(*************************** 647**************************************)
// Wyspa 647 - podajnik opakowań
QABPneumatic647ValveCoils[1].0 := P08_CapSorter.QbCapSorterDragActuator;     //[710, 5/3, wysunięcie wideł]
QABPneumatic647ValveCoils[1].1 := NOT P08_CapSorter.QbCapSorterDragActuator;					
QABPneumatic647ValveCoils[1].2 := P08_CapSorter.QbCapSorterDragLeadBefore1Actuator;    //[720, 5/3 , wysunięcie prowaadzenie ]
QABPneumatic647ValveCoils[1].3 := NOT P08_CapSorter.QbCapSorterDragLeadBefore1Actuator;
QABPneumatic647ValveCoils[1].4 := P08_CapSorter.QbCapSorterStoperActuator;   //[730, 5/2, wysunięcie amortyzatora]
QABPneumatic647ValveCoils[1].5;
QABPneumatic647ValveCoils[1].6 := P08_CapSorter.QbCapSorterDragLeadAfter1Actuator;
QABPneumatic647ValveCoils[1].7 := NOT P08_CapSorter.QbCapSorterDragLeadAfter1Actuator;
QABPneumatic647ValveCoils[2].0;
QABPneumatic647ValveCoils[2].1 := QbBlowBeforeGripperScrewer;//nie ma
QABPneumatic647ValveCoils[2].2 := QbGripperScrewerGateBeforeActuator; //nie ma
QABPneumatic647ValveCoils[2].3;
(*********************Koniec 647 **************************************)

(*************************** 641 **************************************)
QABPneumaticPI641ValveCoils[1].0	:= NOT P01_pucksInserter.QbPucksInserterHammer;
QABPneumaticPI641ValveCoils[1].1	:= P01_pucksInserter.QbPucksInserterHammer;					
QABPneumaticPI641ValveCoils[1].2	:= P01_pucksInserter.QbPucksInserterTray;
QABPneumaticPI641ValveCoils[1].3	:= NOT P01_pucksInserter.QbPucksInserterTray;
QABPneumaticPI641ValveCoils[1].4	:= NOT P01_pucksInserter.QbPucksInserterGate1;
QABPneumaticPI641ValveCoils[1].5	:=  P01_pucksInserter.QbPucksInserterGate1;
QABPneumaticPI641ValveCoils[1].6	:=  NOT P01_pucksInserter.QbPucksInserterGate2;
QABPneumaticPI641ValveCoils[1].7	:=  P01_pucksInserter.QbPucksInserterGate2;
QABPneumaticPI641ValveCoils[2].0 	:=  NOT P01_pucksInserter.QbPucksInserterFormGate;
QABPneumaticPI641ValveCoils[2].1	:=  P01_pucksInserter.QbPucksInserterFormGate;
QABPneumaticPI641ValveCoils[2].2	:=  NOT P01_pucksInserter.QbPucksInserterFormPositioning;
QABPneumaticPI641ValveCoils[2].3  :=  FALSE;//:= NOT P01_PucksInserter.QbPucksInserterPushTable_Gate;    //Vasyl 27.05 [670, 5/2 Szlabany stołu podającego]                    
QABPneumaticPI641ValveCoils[2].4	;//:= 	P01_PucksInserter.QbPucksInserterPushTable_Gate;	
QABPneumaticPI641ValveCoils[2].5;
QABPneumaticPI641ValveCoils[2].6	;//:= P01_PucksInserter.QbPucksInserterPushTable_Pushers; //Vasyl 04.08   [5/2 Popychacze stołu podającego]
QABPneumaticPI641ValveCoils[2].7;
(*********************Koniec 641 **************************************)
END_ACTION

ACTION aVTEM:
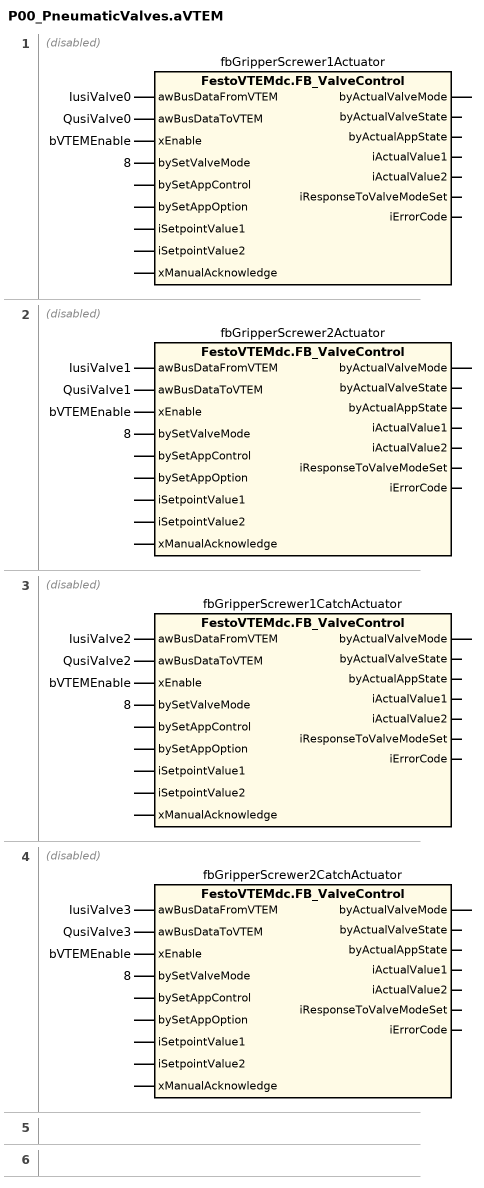
// NETWORK 1 (disabled)
// fbGripperScrewer1Actuator(
//     awBusDataFromVTEM := IusiValve0,
//     awBusDataToVTEM := QusiValve0,
//     xEnable := bVTEMEnable,
//     bySetValveMode := 8); // FestoVTEMdc.FB_ValveControl

// NETWORK 2 (disabled)
// fbGripperScrewer2Actuator(
//     awBusDataFromVTEM := IusiValve1,
//     awBusDataToVTEM := QusiValve1,
//     xEnable := bVTEMEnable,
//     bySetValveMode := 8); // FestoVTEMdc.FB_ValveControl

// NETWORK 3 (disabled)
// fbGripperScrewer1CatchActuator(
//     awBusDataFromVTEM := IusiValve2,
//     awBusDataToVTEM := QusiValve2,
//     xEnable := bVTEMEnable,
//     bySetValveMode := 8); // FestoVTEMdc.FB_ValveControl

// NETWORK 4 (disabled)
// fbGripperScrewer2CatchActuator(
//     awBusDataFromVTEM := IusiValve3,
//     awBusDataToVTEM := QusiValve3,
//     xEnable := bVTEMEnable,
//     bySetValveMode := 8); // FestoVTEMdc.FB_ValveControl

// NETWORK 5

// NETWORK 6
END_ACTION

ACTION aVTEMSignals:
// Wszystkie od 1 do 8 bar
(*
(********VTEM 0********)
(***     F[N]=p[bar]*14,8[N/bar] ************) // od 1,5kg do 12kg
IF lrGripperScrewerPressure = 0 					THEN	lrGripperScrewerPressure := 2; 						END_IF;
IF lrGripperScrewerPressureExhaustLevel < 10	THEN	lrGripperScrewerPressureExhaustLevel := 10;		END_IF;
fbGripperScrewer1Actuator.iSetpointValue2 := (**Smbar Setpoint sir supply pressure during travel**)
ABS(LREAL_TO_INT(((lrGripperScrewerPressure*10)/14.8)*1000));
IF fbGripperScrewer1Actuator.iSetpointValue2 >8000 THEN
	fbGripperScrewer1Actuator.iSetpointValue2 := 8000;
END_IF
IF fbGripperScrewer1Actuator.iSetpointValue2 >8000 THEN
	fbGripperScrewer1Actuator.iSetpointValue2 := 8000;
END_IF
IF P10_GripperScrewer.QbGripperScrewer1Actuator THEN(**Włączanie zaworu**)
	fbGripperScrewer1Actuator.bySetAppControl	:= 2;
	fbGripperScrewer1Actuator.iSetpointValue1	:= LREAL_TO_INT(lrGripperScrewerPressureExhaustLevel*100);//10000;(**Setpoint opening degree axhaust air flow control**)
ELSE
	fbGripperScrewer1Actuator.bySetAppControl	:= 3;
	fbGripperScrewer1Actuator.iSetpointValue1	:= 10000;(**Setpoint opening degree axhaust air flow control**)
END_IF	
IF fbGripperScrewer1Actuator.iResponseToValveModeSet = 1037 (*Acknoledge_needed*) THEN
	fbGripperScrewer1Actuator.xManualAcknowledge := TRUE;	ELSE
	fbGripperScrewer1Actuator.xManualAcknowledge := FALSE;	END_IF
	
	
(********VTEM 1********)
(***     F[N]=p[bar]*14,8[N/bar] ************) // od 1,5kg do 12kg
IF lrGripperScrewerPressure = 0 					THEN	lrGripperScrewerPressure := 2; 						END_IF;
IF lrGripperScrewerPressureExhaustLevel < 10	THEN	lrGripperScrewerPressureExhaustLevel := 10;		END_IF;
fbGripperScrewer2Actuator.iSetpointValue2 := (**Smbar Setpoint sir supply pressure during travel**)
ABS(LREAL_TO_INT(((lrGripperScrewerPressure*10)/14.8)*1000));
IF fbGripperScrewer2Actuator.iSetpointValue2 >8000 THEN
	fbGripperScrewer2Actuator.iSetpointValue2 := 8000;
END_IF
IF fbGripperScrewer2Actuator.iSetpointValue2 >8000 THEN
	fbGripperScrewer2Actuator.iSetpointValue2 := 8000;
END_IF
IF P10_GripperScrewer.QbGripperScrewer2Actuator THEN(**Włączanie zaworu**)
	fbGripperScrewer2Actuator.bySetAppControl	:= 2;
	fbGripperScrewer2Actuator.iSetpointValue1	:= LREAL_TO_INT(lrGripperScrewerPressureExhaustLevel*100);(**Setpoint opening degree axhaust air flow control**)
ELSE
	fbGripperScrewer2Actuator.bySetAppControl	:= 3;
	fbGripperScrewer2Actuator.iSetpointValue1	:= 10000;(**Setpoint opening degree axhaust air flow control**)
END_IF	
IF fbGripperScrewer2Actuator.iResponseToValveModeSet = 1037 (*Acknoledge_needed*) THEN
	fbGripperScrewer2Actuator.xManualAcknowledge := TRUE;	ELSE
	fbGripperScrewer2Actuator.xManualAcknowledge := FALSE;	END_IF
	
	
(********VTEM 2********)
IF lrGripperScrewerPressure = 0 					THEN	lrGripperScrewerPressure := 3; 						END_IF;
IF (lrGripperScrewerCatchPressureExhaustLevel < 10)	THEN	lrGripperScrewerCatchPressureExhaustLevel := 10;		END_IF; // bylo <1000
fbGripperScrewer1CatchActuator.iSetpointValue2 := (**Smbar Setpoint sir supply pressure during travel**)
ABS(LREAL_TO_INT(((lrGripperScrewerPressure*10)/26.2)*1000));
IF fbGripperScrewer1CatchActuator.iSetpointValue2 >8000 THEN
	fbGripperScrewer1CatchActuator.iSetpointValue2 := 8000;
END_IF
IF P10_GripperScrewer.QbGripperScrewer1CatchActuator THEN(**Włączanie zaworu**)
	fbGripperScrewer1CatchActuator.bySetAppControl	:= 1;
	fbGripperScrewer1CatchActuator.iSetpointValue1	:= LREAL_TO_INT((lrGripperScrewerCatchPressureExhaustLevel*15.5)-55);(**Setpoint opening degree axhaust air flow control**)
ELSE
	fbGripperScrewer1CatchActuator.bySetAppControl	:= 2;
	fbGripperScrewer1CatchActuator.iSetpointValue1	:= 10000;(**Setpoint opening degree axhaust air flow control**)
END_IF
IF fbGripperScrewer1CatchActuator.iResponseToValveModeSet = 1037 (*Acknoledge_needed*) THEN
	fbGripperScrewer1CatchActuator.xManualAcknowledge := TRUE;	ELSE
	fbGripperScrewer1CatchActuator.xManualAcknowledge := FALSE;	END_IF	
		
	
(********VTEM 3********)
IF lrGripperScrewerPressure = 0 					THEN	lrGripperScrewerPressure := 3; 						END_IF;
IF ((lrGripperScrewerCatchPressureExhaustLevel) < 10)	THEN	lrGripperScrewerCatchPressureExhaustLevel := 10;		END_IF; // było <1000 i 100000

fbGripperScrewer2CatchActuator.iSetpointValue2 := (**Smbar Setpoint sir supply pressure during travel**)
ABS(LREAL_TO_INT(((lrGripperScrewerPressure*10)/26.2)*1000));
IF fbGripperScrewer2CatchActuator.iSetpointValue2 >8000 THEN
	fbGripperScrewer2CatchActuator.iSetpointValue2 := 8000;
END_IF
IF P10_GripperScrewer.QbGripperScrewer2CatchActuator THEN(**Włączanie zaworu**)
	fbGripperScrewer2CatchActuator.bySetAppControl	:= 1;
	fbGripperScrewer2CatchActuator.iSetpointValue1	:= LREAL_TO_INT((lrGripperScrewerCatchPressureExhaustLevel*15.5)-55);(**Setpoint opening degree axhaust air flow control**)
ELSE
	fbGripperScrewer2CatchActuator.bySetAppControl	:= 2;
	fbGripperScrewer2CatchActuator.iSetpointValue1	:= 10000;(**Setpoint opening degree axhaust air flow control**)
END_IF
IF fbGripperScrewer2CatchActuator.iResponseToValveModeSet = 1037 (*Acknoledge_needed*) THEN
	fbGripperScrewer2CatchActuator.xManualAcknowledge := TRUE;	ELSE
	fbGripperScrewer2CatchActuator.xManualAcknowledge := FALSE;	END_IF	
			
	
*)
END_ACTION

END_PROGRAM

// ---- POUs/FB/Various/FB_4_20mA_TO_INT.TcPOU
FUNCTION_BLOCK FB_4_20mA_TO_INT
VAR_INPUT
	iIN		:	INT;	(*Zmienna skalowana*)
	rXmin	:	REAL;	(*Dolny zakres zmiennej przeskalowanej*)
	rXmax	:	REAL;	(*Górny zakres zmiennej przeskalowanej*)
	rYmin	:	REAL;	(*Dolny zakres zmiennej skalowanej*)
	rYmax	:	REAL;	(*Górny zakres zmiennej skalowanej*)
END_VAR
VAR_OUTPUT
	bError  :	BOOL;
	iOUT	:	INT;	(*Zmienna skalowana*)
END_VAR
VAR
	rfA		:	REAL;	
	rfB		:	REAL;	
	rfC		:	REAL;	
END_VAR


rfA := (rYmax-rYmin)/(rXmax-rXmin);
rfB := (INT_TO_REAL(iIN)-rXmin);
rfC := rYmin;
iOUT := REAL_TO_INT(rfA*rfB+rfC);

IF iIN < rXmin-1 OR iIN>rXmax+1 THEN
	bError	:= TRUE;
	iOUT	:= REAL_TO_INT(rYmax);
ELSE
	bError	:= FALSE;
END_IF

END_FUNCTION_BLOCK

// ---- POUs/FB/Conversions/BitOriented/F_2Bytes_To_Word.TcPOU
(****************************************************************************************)
(*							Beckhoff Automation Poland									*)
(*								F_2Bytes_To_Word v1.0									*)
(*									15.02.2010											*)
(*		Funkcja tworząca zmienną typu WORD z dwóch zmiennych typu BYTE					*)
(*______________________________________________________________________________________*)
FUNCTION F_2Bytes_To_Word : WORD
VAR_INPUT
	byHigh	:	BYTE;
	byLow	:	BYTE;
END_VAR
VAR
END_VAR

F_2Bytes_To_Word := byHigh;
F_2Bytes_To_Word := SHL(F_2Bytes_To_Word,8);
F_2Bytes_To_Word := F_2Bytes_To_Word + byLow;

END_FUNCTION

// ---- POUs/P10_GripperScrewer.TcPOU
(*
Nazwa:			P10_GripperScrewer
Opis:			Stacja zakecarki szczekowej
Wersja:			v0.2
Data:			2018-10-10
Autor:			DP
Urzadzenia:		
Konfiguracja:	
Info:
- aktualizacja bloków
*)
PROGRAM P10_GripperScrewer
VAR_INPUT
	IlrGripperScrewer1HeightCV 							: LREAL;		// Wejscie czujnika dociśnięcia
	IlrGripperScrewer2HeightCV 							: LREAL;		// Wejscie czujnika dociśnięcia
	IbGripperScrewer1CatchActuatorSensor 		  		: BOOL;			// Czujnik otwarcia 
	IbGripperScrewer2CatchActuatorSensor 		  		: BOOL;			// Czujnik otwarcia
	{warning {'dodac czujniki otwarcia chwytaka'}
	IbGripperScrewersThirdFormCheckFormSensor	 	AT %I*	: BOOL; 		// Czujnik dojazdu 3 formatki
	IbGripperScrewersBeforeThirdFormCheckFormSensor	AT %I* 	: BOOL; 		// Czujnik po 3 formatce
	IbGripperScrewersSixthFormCheckFormSensor 		AT %I*	: BOOL;			//Czujnik dojazdu 6 formatki
	IbGripperScrewersDragUpSensor 			 		AT %I*	: BOOL;			// Czujnik
	IbGripperScrewersDragDownSensor 			 	AT %I*	: BOOL;			// Czujnik
	IbGripperScrewersDragHomingSensor 				AT %I*	: BOOL;			// Czujnik bazowania
	IbGripperScrewersDragLeadBefore1UpSensor 		AT %I* 	: BOOL;			// Czujnik
	IbGripperScrewersDragLeadBefore2UpSensor 		AT %I* 	: BOOL;			// Czujnik
END_VAR
VAR
	tonSimu1											:	ton;
	tonSimu2											:	ton;
	//ZMIENNE ZAKRĘCARKI	
	fb2GripperScrewer1									: FB_2GripperScrewers; 				// Blok funkcyjny sterujący zakręcarką szczękową
	fb2GripperScrewerNew1								: FB_2GripperScrewers_New; 			// Blok funkcyjny sterujący zakręcarką szczękową
	eGripperScrewer1State								: E_Station;						// Stan zakręcarki
	eGripperScrewer1RunningState						: E_GripperScrewer;				// Stan zakręcarki
	fb2GripperScrewer2									: FB_2GripperScrewers; 				// Blok funkcyjny sterujący zakręcarką szczękową
	fb2GripperScrewerNew2								: FB_2GripperScrewers_New; 			// Blok funkcyjny sterujący zakręcarką szczękową
	eGripperScrewer2State								: E_Station;						// Stan zakręcarki
	eGripperScrewer2RunningState						: E_GripperScrewer;				// Stan zakręcarki
	fbGripperScrewer1State								: FB_State;
	fbGripperScrewer2State								: FB_State;
	                                        		
	//Zmienne chwytaka                      		
	fbGripperScrewer1CatchStation						: FB_CatchStation;			// Blok funkcyjny sterowania chwytaka zakręcarką szczękową
	eGripperScrewer1CatchState							: E_Station;                  // Stan chwytaka stabilizujšcego pod zakręcarkš
	eGripperScrewer1CatchRunningState					: E_CatchStationState;        // Stan chwytaka stabilizujšcego pod zakręcarkš
	fbGripperScrewer1CatchState							: FB_State;
	
	//WEJSCIA WYJSCIA
	QbGripperScrewer1Actuator							: BOOL; 				// Sterowanie siłownikiem chwytaka zakrecarki szczękowej (Podłączenie do Bajtu sterującego wyspy)
	QnGripperScrewer1TorqueLimit 				AT %Q*	: UINT; 				// Ograniczenie momentu napędu zakręcarki szczękowej 
	QnGripperScrewer1ProportionalGain 			AT %Q*	: REAL; 				// Kp 
	IdiGripperScrewer1HeightCV 					AT %I*	: DINT;			// Wejscie czujnika dociśnięcia
	IrGripperScrewer1ActualMotorTemperature 	AT %I*	: REAL; 				// Aktualna temperatura silnika zakręcarki
	
	//Chwytak zakecarki szczękowej
	QbGripperScrewer1CatchHeightUpCmd 			AT %Q*	: BOOL; 				// Wyjście sterujące podnośnikiem siłownika stabilizującego pod zakręcarką szczękową, Silnik w górę
	QbGripperScrewer1CatchHeightDownCmd 		AT %Q*	: BOOL; 				// Wyjście sterujące podnośnikiem siłownika stabilizującego pod zakręcarką szczękową, Silnik w dół
	QbGripperScrewer1CatchActuator						: BOOL; 				// Sterowanie siłownikiem chwytaka stabilizującego pod zakręcarką szczękową (Podłączenie do Bajtu sterującego wyspy)
	IbGripperScrewer1CatchHeightEncoderPulse 	AT %I*  : BOOL;					// Wejście impulsów enkodera podnośnika chwytaka pod zakręcarką
	
	tofTimerGripperScrewer1Enable						: TOF;
	rtbGripperScrewer12EnableShow						: R_TRIG;
	ftbGripperScrewer12EnableShow						: F_TRIG;	
	rtEnable1											: R_TRIG;
	
	(*Wykres dozowania*)
	fbGripperScrewer1Chart								: FB_WriteDataToArrayString;
	fbGripperScrewer1StChart							: FB_WriteDataToArrayOfArrays;
	fbGripperScrewer2StChart							: FB_WriteDataToArrayOfArrays;
	rtStartGripper1Screwing								: R_TRIG;
	lrGripperScrewer1AxisStartPosition					: LREAL;
	nCountTest555										: INT;
	nCountTest556										: INT;
	nCountTest557										: INT;
	nGripperScrewer1AdjustingDialog						: INT;
	bGripperScrewer1AdjustTorqueDialog					: BOOL;
	nTstcount											: INT;

	//Zmienne chwytaka
	fbGripperScrewer2CatchStation						: FB_CatchStation;			// Blok funkcyjny sterowania chwytaka zakręcarką szczękową
	eGripperScrewer2CatchState							: E_Station;                  // Stan chwytaka stabilizujšcego pod zakręcarkš
	eGripperScrewer2CatchRunningState					: E_CatchStationState;        // Stan chwytaka stabilizujšcego pod zakręcarkš
	fbGripperScrewerCatch2State							: FB_State;
	
	
	//WEJSCIA WYJSCIA
	QbGripperScrewer2Actuator							: BOOL; 	(*Pneu*)		// Sterowanie siłownikiem chwytaka zakrecarki szczękowej (Podłączenie do Bajtu sterującego wyspy)
	QnGripperScrewer2TorqueLimit 				AT %Q*	: UINT; 	(*do driva*)	// Ograniczenie momentu napędu zakręcarki szczękowej 
	QnGripperScrewer2ProportionalGain 			AT %Q*	: REAL; 				// Kp 
	IrGripperScrewer2ActualMotorTemperature 	AT %I*	: REAL; 	(*do driva*)	// Aktualna temperatura silnika zakręcarki
	IdiGripperScrewer2HeightCV 					AT %I*	: DINT;			// Wejscie czujnika dociśnięcia
	IbGripperScrewersHeightEncoderSetCDone				AT %I*: BOOL;
	IudiGripperScrewersHeightEncoderCV          AT %I*: UDINT;
	QbGripperScrewersHeightEncoderSetC 			AT %Q*: BOOL;
	QudiGripperScrewersHeightEncoderSetCV       AT %Q*: UDINT;
	
	//Chwytak zakecarki szczękowej
	QbGripperScrewer2CatchHeightUpCmd 			AT %Q*	: BOOL; 			(*PLC.A19*)	 	// Wyjście sterujące podnośnikiem siłownika stabilizującego pod zakręcarką szczękową, Silnik w górę
	QbGripperScrewer2CatchHeightDownCmd 		AT %Q*	: BOOL; 		(*PLC.A19*)		// Wyjście sterujące podnośnikiem siłownika stabilizującego pod zakręcarką szczękową, Silnik w dół
	QbGripperScrewer2CatchActuator						: BOOL; 					(*Pneu*)		// Sterowanie siłownikiem chwytaka stabilizującego pod zakręcarką szczękową (Podłączenie do Bajtu sterującego wyspy)
	IbGripperScrewer2CatchHeightEncoderPulse  	AT %I*  : BOOL;	(*PLC.A15*)		// Wejście impulsów enkodera podnośnika chwytaka pod zakręcarką

	tofTimerGripperScrewer2Enable						: TOF;


	(*Wykres dozowania*)
	fbGripperScrewer2Chart								: FB_WriteDataToArrayString;
	rtStartGripper2Screwing								: R_TRIG;
	lrGripperScrewer2AxisStartPosition					: LREAL;
	
	(*******PRZECIAGANIE**********)
	fbGripperScrewersDragStation						: FB_FormsDragStepper;
	eFormsDragingPneumaticState							: E_Station;						// Stan zakręcarki
	eFormsDragingPneuamticRunningState					: E_DragStationState;			// Stan zakręcarki
	fbFormsDragingPneumaticState						: FB_State;
	
	//WEJSCIA I WYJSCIA SPRZETOW
	QbGripperScrewersDragLeadBefore1Actuator        	:BOOL;						// Siłownikiem prowadzenia przed 1(1 faza)
	QbGripperScrewersDragActuator                	  	:BOOL;						// Siłownikiem przeciągania (1 faza)
	
	tDelayCatchValve									: TIME;
	tonGriperScrewerCatch1ValveOpenSensor				: TON;
	tonGriperScrewerCatch2ValveOpenSensor				: TON;
		
	(*kasowanie offsetu*)
	tonGripperScrewer1SetPositionOffsetReset			: TON;
	tonGripperScrewer2SetPositionOffsetReset			: TON;

	(*Filtrowqanie momentu*)
	fbFilterTorque1						: FB_FilterEx;					// Bloczek do filtrowania (*NOWE*)
	rFilteredTorque1Value				: REAL;							// Zmiena odfiltrowana (*NOWE*)
	fbFilterTorque2						: FB_FilterEx;					// Bloczek do filtrowania (*NOWE*)
	rFilteredTorque2Value				: REAL;							// Zmiena odfiltrowana (*NOWE*)
	
	(*Szukanie gwintu*)
	lrGripperScrewerPushingCapPositionTemp	:	LREAL;
	lrGripperScrewerScrewingCapPositionTemp	:	LREAL;
	rtGripperScrewerFindScrewAdjust			:	R_TRIG;
	rtGripperScrewerOption5					:	R_TRIG;
	iGripperScrewerFindScrewAdjust			:	INT;
	
	(*smieci*)
	btemp												: BOOL;
	atemp1												: AXIS_REF;
	atemp2												: AXIS_REF;
	
	(*inne*)
	bSimulationGripper									: BOOL;

	tofTimerGripperScrewer1Catch: TOF;
	tofTimerGripperScrewer2Catch: TOF;
	
//dodatkowa obsługa stopera formatek przy dojeździe 
	

	//tpStoperTimerOn							:TP;	// timer do generowania impulsu
	//fbStoperSensorDelay						:FB_InputFilter;	// filtr do generowania sygnału 
	//tofQbGripperScrewerStoperActuator		:TOF;
	//lrStoperPosition: LREAL;
	bTestZakrecania: BOOL;
	
	rtfb2GripperScrewer1Done: R_TRIG;
	rtfb2GripperScrewer2Done: R_TRIG;	

	iGripperScrewer1Info1 : INT;
	iGripperScrewer2Info1 : INT;
	iGripperScrewer1NoWarningInRow : INT;
	iGripperScrewer2NoWarningInRow : INT;	
	bGripperScrewer1ChangeRubbers :BOOL;
	bGripperScrewer2ChangeRubbers :BOOL;	
	tonbGripperScrewer1ChangeRubbers: TON;
	tonbGripperScrewer2ChangeRubbers: TON;	
	
	//ManualStoper
	rtManualMode	: R_TRIG;
	ftManualMode	: F_TRIG;	
	bGripperScrewerStoperActuatorLastState	:BOOL;
	
	

	
END_VAR

(**Symulacja czujników otwarcia-zamknięcia chwytaka***)

tDelayCatchValve														:=T#50MS;

tonGriperScrewerCatch1ValveOpenSensor(IN:= NOT QbGripperScrewer1CatchActuator, PT:=tDelayCatchValve);
tonGriperScrewerCatch2ValveOpenSensor(IN:= NOT QbGripperScrewer2CatchActuator, PT:=tDelayCatchValve);
aStoper();
aDraging();
aCatch();
aLimits();
aFilter();
aGripperScrewerEnable();
aGripperScrewer();			//Nowa wersja zakrecarek STARA aGripperScrewer();
aGripperScrewerChartHMI();
aGripperScrewerDialogBox();
aGripperScrewerWarnings();
aFindScrewAdjust();
aInfo();

(***Skalownaie wartości zadanej na 1-100%************)
IF lrBottleDragingStationVelocity <50 THEN
	lrBottleDragingStationVelocity	:= 50;
END_IF 

(*** SKALOWANIE WARTOŚCI ZAKRĘCANIA Z Nm na % ***)
IF iPackageCapDiameter = 0 THEN
	iPackageCapDiameter 												:= 20;
END_IF

VIS.iPackageCapDiameterShow;
fb2GripperScrewer1.iScrewer1SetTorque 									:= LREAL_TO_INT((lrGripperScrewingTightTorque/1.5)*100);
fb2GripperScrewer2.iScrewer1SetTorque 									:= LREAL_TO_INT((lrGripperScrewing2TightTorque/1.5)*100);

(*** KONIEC SKALOWANIE WARTOŚCI ZAKRĘCANIA Z Nm na % ***)

(**** SKALOWANIE CZUJNIKOW WYSOKOSCI***)
IdiGripperScrewer1HeightCV;
//fb2GripperScrewer1.lrSpringHeightCV:= (IdiGripperScrewer1HeightCV *-1 ) + 110000;
//fb2GripperScrewer1.lrSpringHeightCV:= TO_LREAL(IdiGripperScrewer1HeightCV) /(-1000.0)+52.5; 
//

IdiGripperScrewer2HeightCV;
//fb2GripperScrewer2.lrSpringHeightCV:= (IdiGripperScrewer2HeightCV *-1 ) + 110000;
//fb2GripperScrewer2.lrSpringHeightCV:= TO_LREAL(IdiGripperScrewer2HeightCV) /(-1000.0)+52.1; 


(* BAZOWANIE - ZMIAN*)

tofTimerGripperScrewer1Catch(IN:=bGripperScrewer1Enable (*AND NOT bChangeover*), PT:=T#8S); 
tofTimerGripperScrewer2Catch(IN:=bGripperScrewer2Enable (*AND NOT bChangeover*), PT:=T#8S); 

rtEnable1(CLK:=fb2GripperScrewer1.bEnable1 OR fb2GripperScrewer2.bEnable1 ,Q=>);

VIS.lrGripperScrewer1LiftActPos											:= aGripperScrewer1LiftAxisRef.NcToPlc.ActPos;
VIS.lrGripperScrewer2LiftActPos											:= aGripperScrewer2LiftAxisRef.NcToPlc.ActPos;


IF rtEnable1.Q AND (P00_PackML.fbPMLAuto.ePMLState = E_PMLState.ePMLState_IDLE OR P00_PackML.fbPMLAuto.ePMLState = E_PMLState.ePMLState_EXECUTE)  THEN
	VIS.bGripperScrewerCatchHeightSet									:= TRUE;
	nCountTest555														:= nCountTest555+1;
ELSIF (fbGripperScrewer1CatchStation.eState=E_Station.eHomingDone AND fbGripperScrewer2CatchStation.eState=E_Station.eHomingDone)  AND fb2GripperScrewer1.eState=E_Station.eHomingDone AND fb2GripperScrewer2.eState=E_Station.eHomingDone THEN
	VIS.bGripperScrewerCatchHeightSet									:= FALSE;
	
ELSIF (fbGripperScrewer1CatchStation.eState=E_Station.eHomingDone AND fbGripperScrewer2CatchStation.eState=E_Station.eHomingDone)  THEN
	VIS.bGripperScrewerHeightSet										:= TRUE;
	
ELSIF (fb2GripperScrewer1.eState=E_Station.eHomingDone AND fb2GripperScrewer2.eState=E_Station.eHomingDone) OR VIS.bErrorOccure THEN
 	VIS.bGripperScrewerHeightSet										:= FALSE;
	nCountTest556														:= nCountTest556+1;
	
ELSIF (fbGripperScrewer1CatchStation.eState=E_Station.eHomingDone AND fbGripperScrewer2CatchStation.eState=E_Station.eHomingDone ) OR VIS.bErrorOccure  THEN
	VIS.bGripperScrewerCatchHeightSet									:= FALSE;
	VIS.bGripperScrewerHeightSet										:= FALSE;	
	nCountTest557														:= nCountTest557+1;
END_IF
(*KONIEC BAZOWANIE - ZMIANA*)


(********* GENEROWANIE STANU STACJI DO WIZKI**********)



fbGripperScrewer1State(
	eState																:= eGripperScrewer1State , 
	bRun																:= VIS.bGripperScrewer1Run OR VIS.bGripperScrewer1Run,	
	eGripperScrewerRunningState											:= eGripperScrewer1RunningState , 
	sStateDesc															=> VIS.sGripperScrewer1State,
	iState																=> VIS.iGripperScrewer1State);
fbGripperScrewer2State(
	eState																:= eGripperScrewer2State , 
	bRun																:= VIS.bGripperScrewer2Run OR VIS.bGripperScrewer2Run,	
	eGripperScrewerRunningState											:= eGripperScrewer2RunningState , 
	sStateDesc															=> VIS.sGripperScrewer2State,
	iState																=> VIS.iGripperScrewer2State);

fbGripperScrewer1CatchState(
	eState																:= eGripperScrewer1CatchState , 
	bRun																:= bGripperScrewer1Catch,	
	eCatchRunningState													:= eGripperScrewer1CatchRunningState , 
	sStateDesc															=> VIS.sGripperScrewerCatch1State,
	iState																=> VIS.iGripperScrewerCatch1State);	
	
fbGripperScrewerCatch2State(
	eState																:= eGripperScrewer2CatchState , 
	bRun																:= bGripperScrewer2Catch,	
	eCatchRunningState													:= eGripperScrewer2CatchRunningState , 
	sStateDesc															=> VIS.sGripperScrewerCatch2State,
	iState																=> VIS.iGripperScrewerCatch2State);	
	
fbFormsDragingPneumaticState(
	eState																:= eFormsDragingPneumaticState , 
	bRun																:= VIS.bBottleDragingStationRun,	
	eFormsDragingRunningState											:= eFormsDragingPneuamticRunningState , 
	sStateDesc															=> VIS.sBottleDragingStationState,
	iState																=> VIS.iBottleDragingStationState);	
	
		
(***** KONIEC GENEROWANIE STANU STACJI DO WIZKI*******)

(******* Wypracowanie sygnałów dla HMI *******)


VIS.bGripperScrewerCatch1ManualActuator;
(********KASOWANIE ROZKAZÓW CYKLI*********)
IF fb2GripperScrewer1.bCycleDone1 AND bManualMode THEN
	VIS.bGripperScrewer1Run 											:= FALSE;
END_IF
IF fb2GripperScrewer2.bCycleDone1 AND bManualMode THEN
	VIS.bGripperScrewer2Run 											:= FALSE;
END_IF

IF fbGripperScrewersDragStation.bCycleDone AND bManualMode THEN
	VIS.bBottleDragingStationRun 				:= FALSE;
	GVL.bBottleDragingStationPrepareRun			:= FALSE;
END_IF

(*Kasowanie offsetu po czasie*)
tonGripperScrewer1SetPositionOffsetReset(IN:=VIS.bGripperScrewer1SetPositionOffset, PT:=T#2S);
IF tonGripperScrewer1SetPositionOffsetReset.Q THEN
	VIS.bGripperScrewer1SetPositionOffset := FALSE;
END_IF
tonGripperScrewer2SetPositionOffsetReset(IN:=VIS.bGripperScrewer2SetPositionOffset, PT:=T#2S);
IF tonGripperScrewer2SetPositionOffsetReset.Q THEN
	VIS.bGripperScrewer2SetPositionOffset := FALSE;
END_IF
(*****KONIEC KASOWANIA ROZKAZÓW CYKLI*****)

aGripperScrewer1LiftAxisRef.NcToPlc.ActPos;
fb2GripperScrewer2.iToolHeight;

ACTION aCatch:
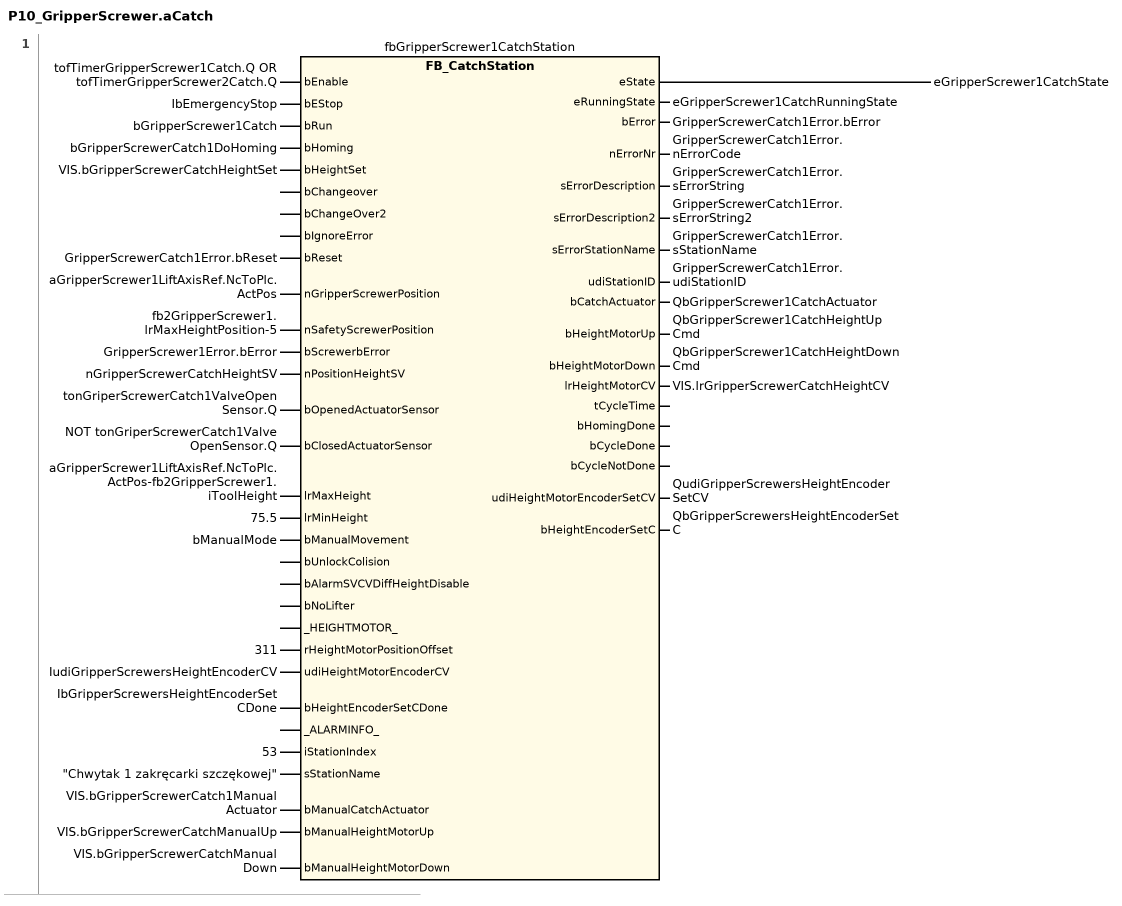
// NETWORK 1
fbGripperScrewer1CatchStation(
    bEnable := tofTimerGripperScrewer1Catch.Q OR tofTimerGripperScrewer2Catch.Q,
    bEStop := IbEmergencyStop,
    bRun := bGripperScrewer1Catch,
    bHoming := bGripperScrewerCatch1DoHoming,
    bHeightSet := VIS.bGripperScrewerCatchHeightSet,
    bReset := GripperScrewerCatch1Error.bReset,
    nGripperScrewerPosition := aGripperScrewer1LiftAxisRef.NcToPlc.ActPos,
    nSafetyScrewerPosition := fb2GripperScrewer1.lrMaxHeightPosition-5,
    bScrewerbError := GripperScrewer1Error.bError,
    nPositionHeightSV := nGripperScrewerCatchHeightSV,
    bOpenedActuatorSensor := tonGriperScrewerCatch1ValveOpenSensor.Q,
    bClosedActuatorSensor := NOT tonGriperScrewerCatch1ValveOpenSensor.Q,
    lrMaxHeight := aGripperScrewer1LiftAxisRef.NcToPlc.ActPos-fb2GripperScrewer1.iToolHeight,
    lrMinHeight := 75.5,
    bManualMovement := bManualMode,
    rHeightMotorPositionOffset := 311,
    udiHeightMotorEncoderCV := IudiGripperScrewersHeightEncoderCV,
    bHeightEncoderSetCDone := IbGripperScrewersHeightEncoderSetCDone,
    iStationIndex := 53,
    sStationName := "Chwytak 1 zakręcarki szczękowej",
    bManualCatchActuator := VIS.bGripperScrewerCatch1ManualActuator,
    bManualHeightMotorUp := VIS.bGripperScrewerCatchManualUp,
    bManualHeightMotorDown := VIS.bGripperScrewerCatchManualDown,
    eRunningState => eGripperScrewer1CatchRunningState,
    bError => GripperScrewerCatch1Error.bError,
    nErrorNr => GripperScrewerCatch1Error.nErrorCode,
    sErrorDescription => GripperScrewerCatch1Error.sErrorString,
    sErrorDescription2 => GripperScrewerCatch1Error.sErrorString2,
    sErrorStationName => GripperScrewerCatch1Error.sStationName,
    udiStationID => GripperScrewerCatch1Error.udiStationID,
    bCatchActuator => QbGripperScrewer1CatchActuator,
    bHeightMotorUp => QbGripperScrewer1CatchHeightUpCmd,
    bHeightMotorDown => QbGripperScrewer1CatchHeightDownCmd,
    lrHeightMotorCV => VIS.lrGripperScrewerCatchHeightCV,
    udiHeightMotorEncoderSetCV => QudiGripperScrewersHeightEncoderSetCV,
    bHeightEncoderSetC => QbGripperScrewersHeightEncoderSetC); // FB_CatchStation
eGripperScrewer1CatchState := fbGripperScrewer1CatchStation.eState;

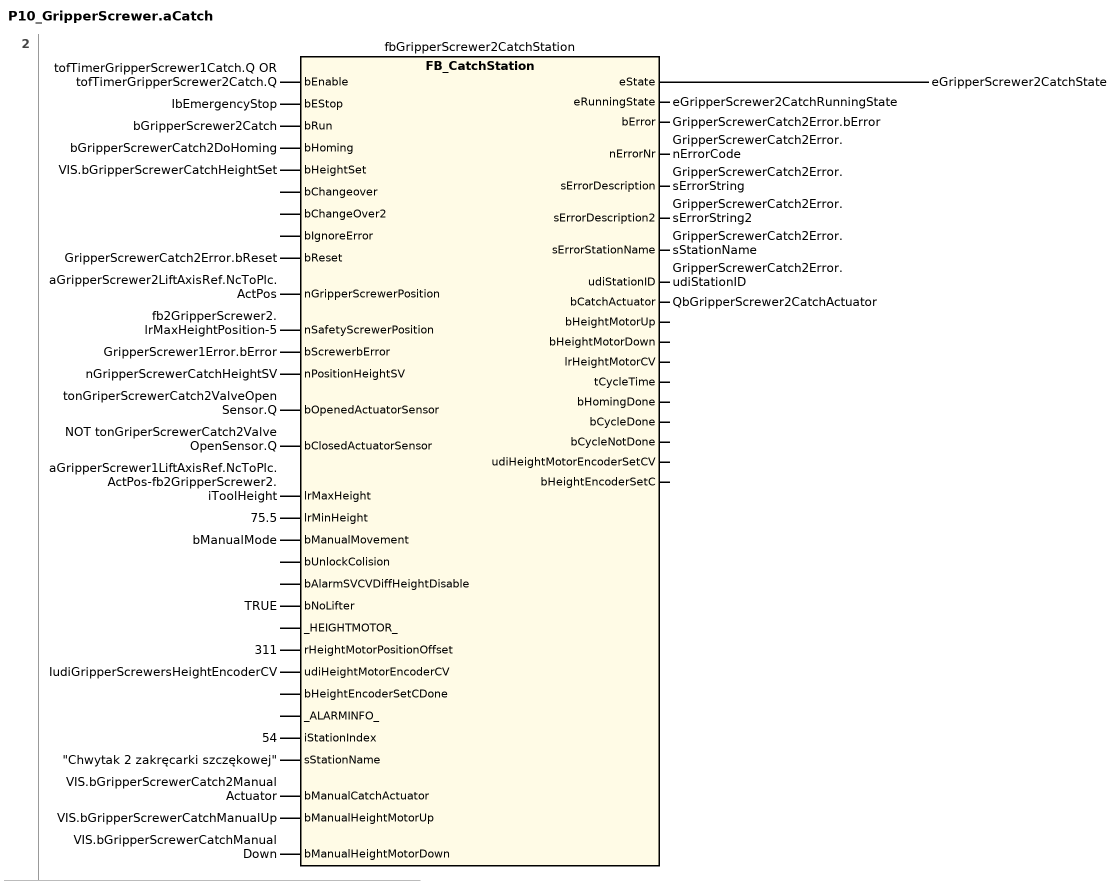
// NETWORK 2
fbGripperScrewer2CatchStation(
    bEnable := tofTimerGripperScrewer1Catch.Q OR tofTimerGripperScrewer2Catch.Q,
    bEStop := IbEmergencyStop,
    bRun := bGripperScrewer2Catch,
    bHoming := bGripperScrewerCatch2DoHoming,
    bHeightSet := VIS.bGripperScrewerCatchHeightSet,
    bReset := GripperScrewerCatch2Error.bReset,
    nGripperScrewerPosition := aGripperScrewer2LiftAxisRef.NcToPlc.ActPos,
    nSafetyScrewerPosition := fb2GripperScrewer2.lrMaxHeightPosition-5,
    bScrewerbError := GripperScrewer1Error.bError,
    nPositionHeightSV := nGripperScrewerCatchHeightSV,
    bOpenedActuatorSensor := tonGriperScrewerCatch2ValveOpenSensor.Q,
    bClosedActuatorSensor := NOT tonGriperScrewerCatch2ValveOpenSensor.Q,
    lrMaxHeight := aGripperScrewer1LiftAxisRef.NcToPlc.ActPos-fb2GripperScrewer2.iToolHeight,
    lrMinHeight := 75.5,
    bManualMovement := bManualMode,
    bNoLifter := TRUE,
    rHeightMotorPositionOffset := 311,
    udiHeightMotorEncoderCV := IudiGripperScrewersHeightEncoderCV,
    iStationIndex := 54,
    sStationName := "Chwytak 2 zakręcarki szczękowej",
    bManualCatchActuator := VIS.bGripperScrewerCatch2ManualActuator,
    bManualHeightMotorUp := VIS.bGripperScrewerCatchManualUp,
    bManualHeightMotorDown := VIS.bGripperScrewerCatchManualDown,
    eRunningState => eGripperScrewer2CatchRunningState,
    bError => GripperScrewerCatch2Error.bError,
    nErrorNr => GripperScrewerCatch2Error.nErrorCode,
    sErrorDescription => GripperScrewerCatch2Error.sErrorString,
    sErrorDescription2 => GripperScrewerCatch2Error.sErrorString2,
    sErrorStationName => GripperScrewerCatch2Error.sStationName,
    udiStationID => GripperScrewerCatch2Error.udiStationID,
    bCatchActuator => QbGripperScrewer2CatchActuator); // FB_CatchStation
eGripperScrewer2CatchState := fbGripperScrewer2CatchStation.eState;
END_ACTION

ACTION aDraging:
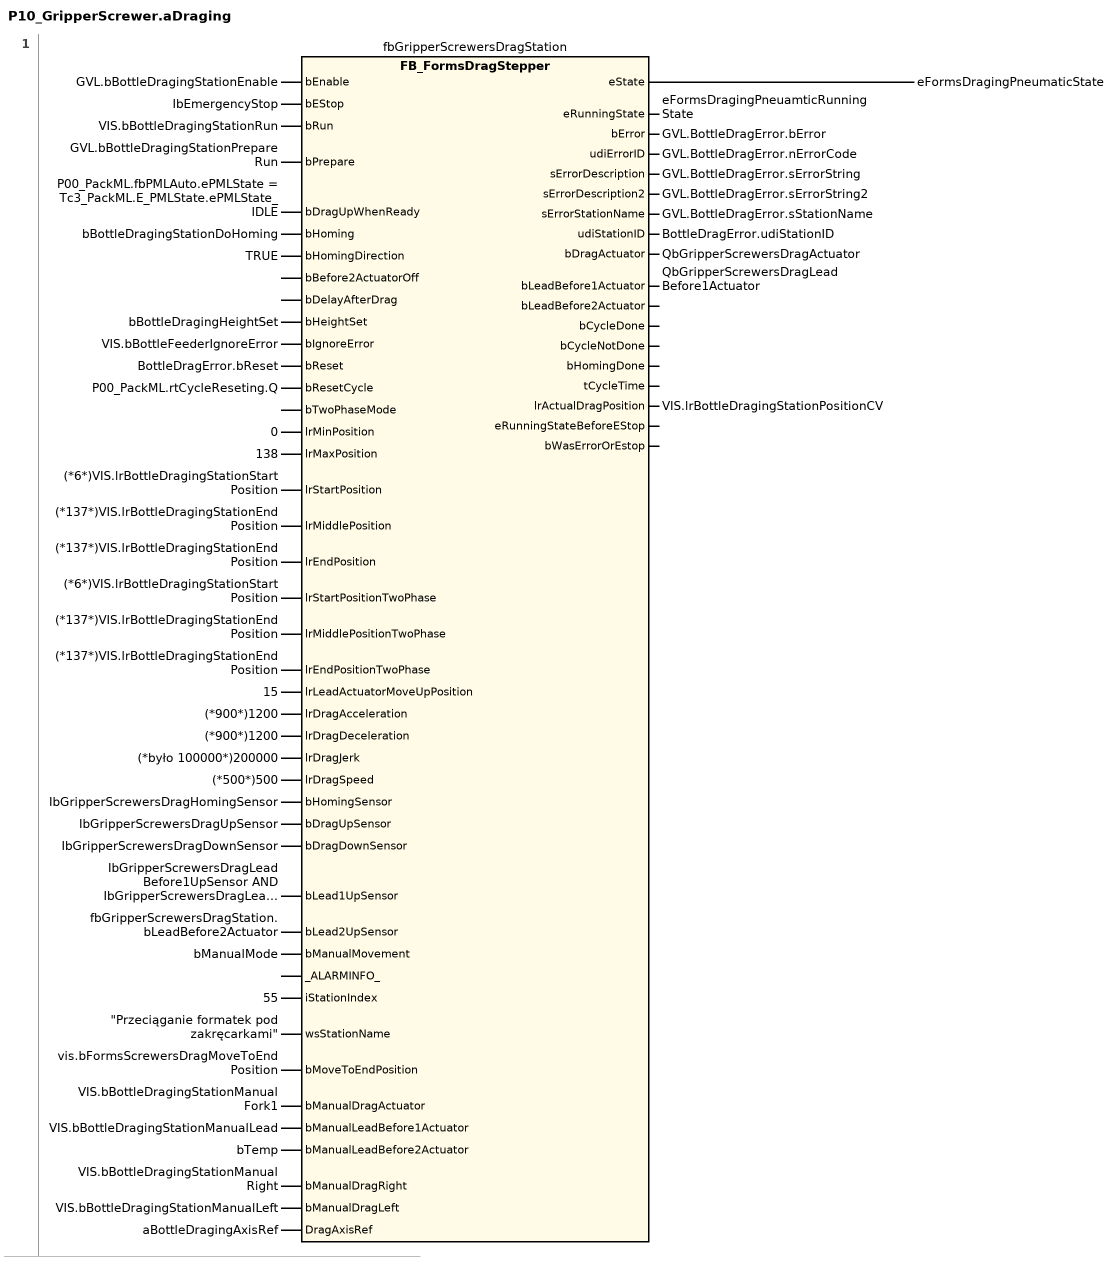
// NETWORK 1
fbGripperScrewersDragStation(
    bEnable := GVL.bBottleDragingStationEnable,
    bEStop := IbEmergencyStop,
    bRun := VIS.bBottleDragingStationRun,
    bPrepare := GVL.bBottleDragingStationPrepareRun,
    bDragUpWhenReady := P00_PackML.fbPMLAuto.ePMLState = Tc3_PackML.E_PMLState.ePMLState_IDLE,
    bHoming := bBottleDragingStationDoHoming,
    bHomingDirection := TRUE,
    bHeightSet := bBottleDragingHeightSet,
    bIgnoreError := VIS.bBottleFeederIgnoreError,
    bReset := BottleDragError.bReset,
    bResetCycle := P00_PackML.rtCycleReseting.Q,
    lrMinPosition := 0,
    lrMaxPosition := 138,
    lrStartPosition := (*6*)VIS.lrBottleDragingStationStartPosition,
    lrMiddlePosition := (*137*)VIS.lrBottleDragingStationEndPosition,
    lrEndPosition := (*137*)VIS.lrBottleDragingStationEndPosition,
    lrStartPositionTwoPhase := (*6*)VIS.lrBottleDragingStationStartPosition,
    lrMiddlePositionTwoPhase := (*137*)VIS.lrBottleDragingStationEndPosition,
    lrEndPositionTwoPhase := (*137*)VIS.lrBottleDragingStationEndPosition,
    lrLeadActuatorMoveUpPosition := 15,
    lrDragAcceleration := (*900*)1200,
    lrDragDeceleration := (*900*)1200,
    lrDragJerk := (*było 100000*)200000,
    lrDragSpeed := (*500*)500,
    bHomingSensor := IbGripperScrewersDragHomingSensor,
    bDragUpSensor := IbGripperScrewersDragUpSensor,
    bDragDownSensor := IbGripperScrewersDragDownSensor,
    bLead1UpSensor := IbGripperScrewersDragLeadBefore1UpSensor AND IbGripperScrewersDragLeadBefore2UpSensor,
    bLead2UpSensor := fbGripperScrewersDragStation.bLeadBefore2Actuator,
    bManualMovement := bManualMode,
    iStationIndex := 55,
    wsStationName := "Przeciąganie formatek pod zakręcarkami",
    bMoveToEndPosition := vis.bFormsScrewersDragMoveToEndPosition,
    bManualDragActuator := VIS.bBottleDragingStationManualFork1,
    bManualLeadBefore1Actuator := VIS.bBottleDragingStationManualLead,
    bManualLeadBefore2Actuator := bTemp,
    bManualDragRight := VIS.bBottleDragingStationManualRight,
    bManualDragLeft := VIS.bBottleDragingStationManualLeft,
    DragAxisRef := aBottleDragingAxisRef,
    eRunningState => eFormsDragingPneuamticRunningState,
    bError => GVL.BottleDragError.bError,
    udiErrorID => GVL.BottleDragError.nErrorCode,
    sErrorDescription => GVL.BottleDragError.sErrorString,
    sErrorDescription2 => GVL.BottleDragError.sErrorString2,
    sErrorStationName => GVL.BottleDragError.sStationName,
    udiStationID => BottleDragError.udiStationID,
    bDragActuator => QbGripperScrewersDragActuator,
    bLeadBefore1Actuator => QbGripperScrewersDragLeadBefore1Actuator,
    lrActualDragPosition => VIS.lrBottleDragingStationPositionCV); // FB_FormsDragStepper
eFormsDragingPneumaticState := fbGripperScrewersDragStation.eState;
END_ACTION

ACTION aFilter:
fbFilterTorque1(
				rIn:=				LREAL_TO_REAL(aGripperScrewer1AxisRef.NcToPlc.ActTorque), 
				tTimeConstant:= 	T#3MS, 
				rOut=>				rFilteredTorque1Value);
fbFilterTorque2(
				rIn:=				LREAL_TO_REAL(aGripperScrewer2AxisRef.NcToPlc.ActTorque), 
				tTimeConstant:= 	T#3MS, 
				rOut=>				rFilteredTorque2Value);
END_ACTION

ACTION aFindScrewAdjust:
bGripperScrewerFindScrewAdjust;
bGripperScrewerOption5;
(*Wykrywanie potrzeby ponownego włączenia szukania wartości MIN i MAX przy zaznaczonej opcji szukania gwintu z czujnikiem wysokości*)
(*Szczególnie po zmianie parametrów wysokości*)
lrGripperScrewerPushingCapPosition;
lrGripperScrewerScrewingCapPosition;

rtGripperScrewerFindScrewAdjust(CLK:=
							bGripperScrewerOption5 AND 
							(
							lrGripperScrewerPushingCapPositionTemp <> lrGripperScrewerPushingCapPosition OR
							lrGripperScrewerScrewingCapPositionTemp <> lrGripperScrewerScrewingCapPosition
							)
							,Q=>);

rtGripperScrewerOption5		(CLK:=		bGripperScrewerOption5,	Q=>);				

IF rtGripperScrewerFindScrewAdjust.Q OR rtGripperScrewerOption5.Q THEN
	bGripperScrewerFindScrewAdjust 				:=	TRUE;
	iGripperScrewerFindScrewAdjust				:=	iGripperScrewerFindScrewAdjust	+	1;
	lrGripperScrewerPushingCapPositionTemp 		:=	lrGripperScrewerPushingCapPosition; 	
	lrGripperScrewerScrewingCapPositionTemp 	:=	lrGripperScrewerScrewingCapPosition;
END_IF
END_ACTION

ACTION aGripperScrewer:
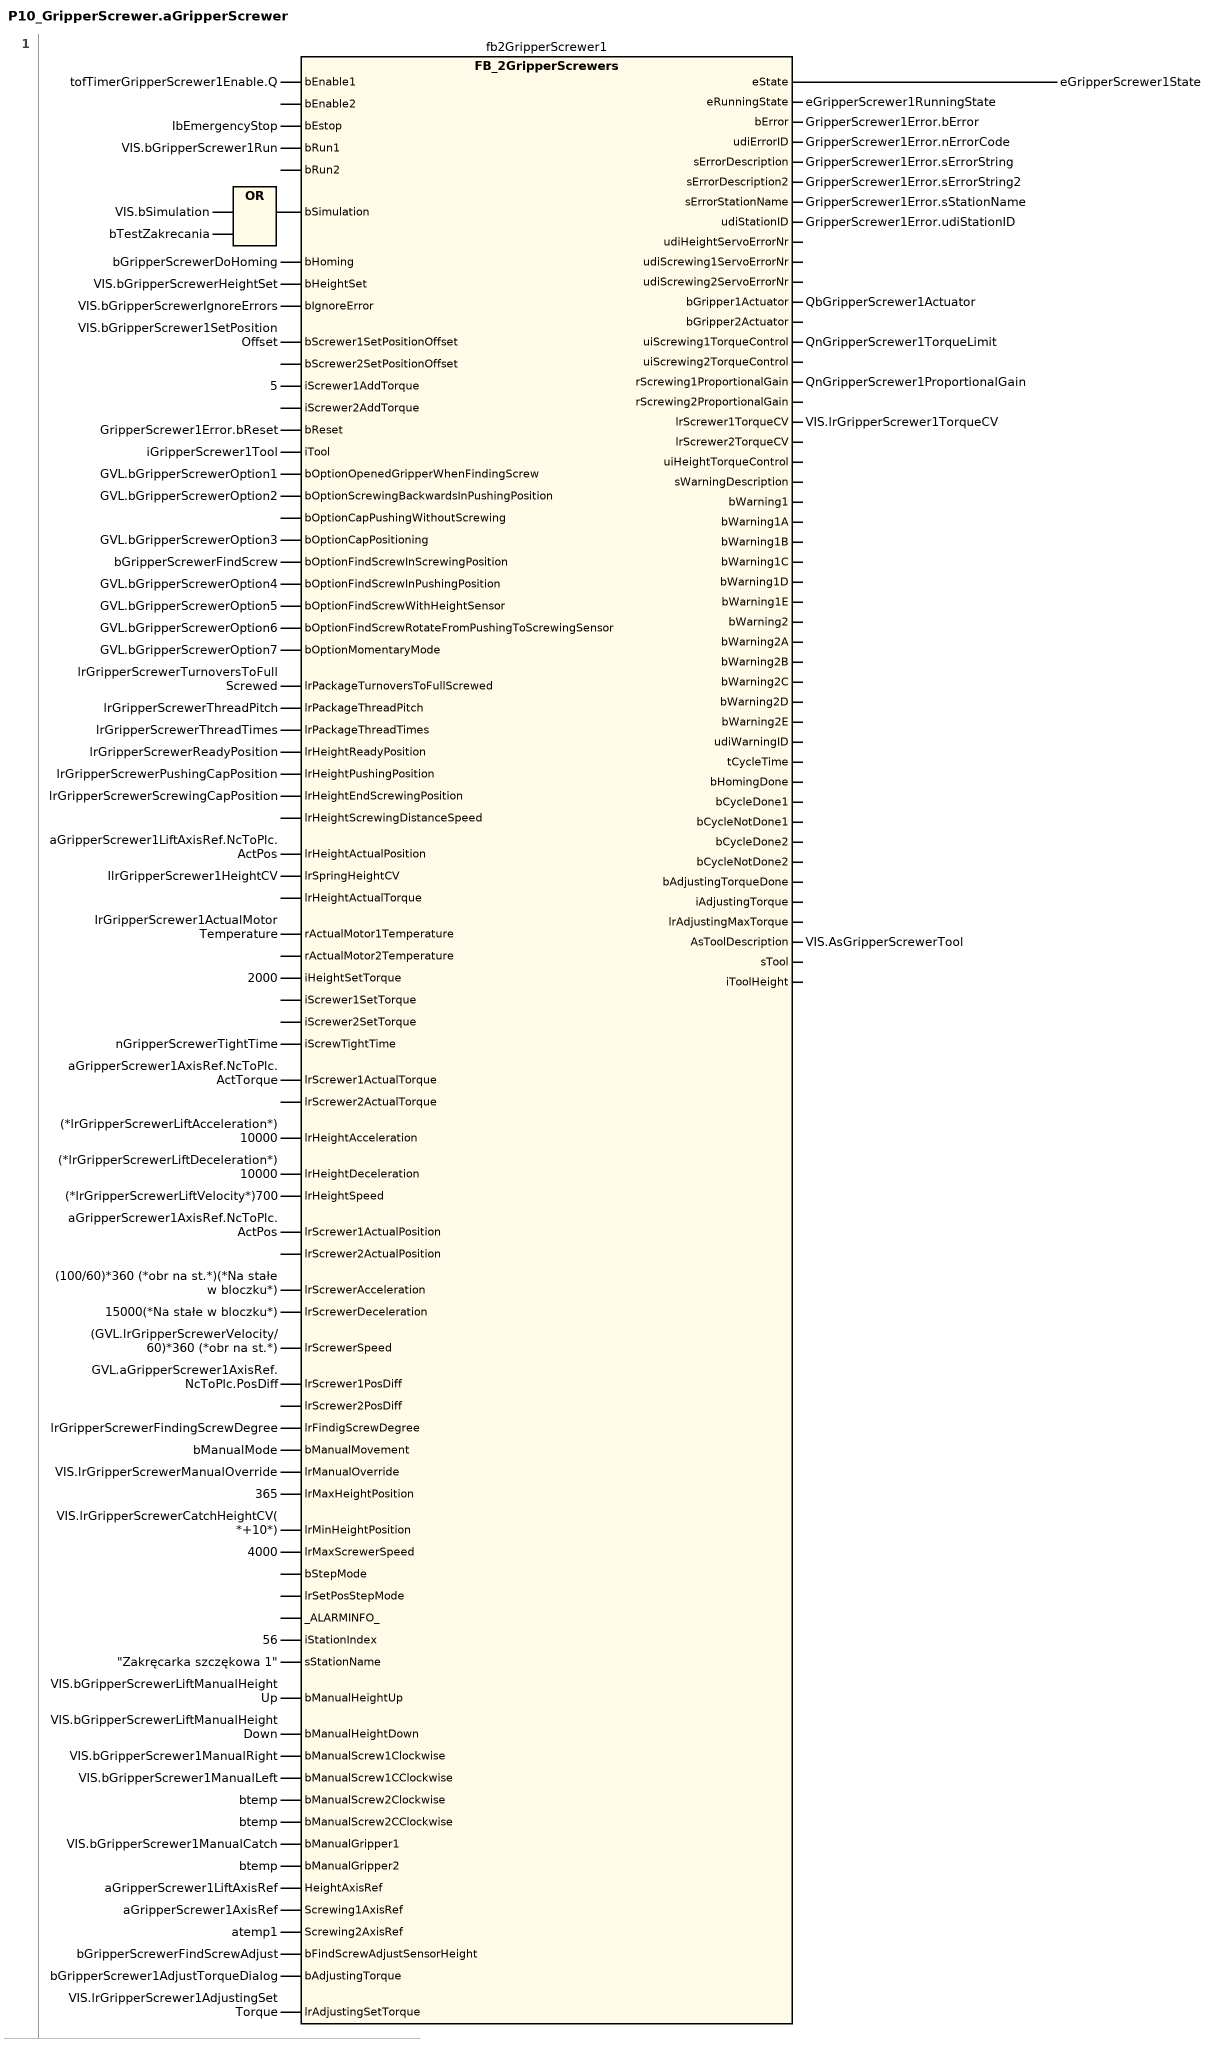
// NETWORK 1
fb2GripperScrewer1(
    bEnable1 := tofTimerGripperScrewer1Enable.Q,
    bEstop := IbEmergencyStop,
    bRun1 := VIS.bGripperScrewer1Run,
    bSimulation := VIS.bSimulation OR bTestZakrecania,
    bHoming := bGripperScrewerDoHoming,
    bHeightSet := VIS.bGripperScrewerHeightSet,
    bIgnoreError := VIS.bGripperScrewerIgnoreErrors,
    bScrewer1SetPositionOffset := VIS.bGripperScrewer1SetPositionOffset,
    iScrewer1AddTorque := 5,
    bReset := GripperScrewer1Error.bReset,
    iTool := iGripperScrewer1Tool,
    bOptionOpenedGripperWhenFindingScrew := GVL.bGripperScrewerOption1,
    bOptionScrewingBackwardsInPushingPosition := GVL.bGripperScrewerOption2,
    bOptionCapPositioning := GVL.bGripperScrewerOption3,
    bOptionFindScrewInScrewingPosition := bGripperScrewerFindScrew,
    bOptionFindScrewInPushingPosition := GVL.bGripperScrewerOption4,
    bOptionFindScrewWithHeightSensor := GVL.bGripperScrewerOption5,
    bOptionFindScrewRotateFromPushingToScrewingSensor := GVL.bGripperScrewerOption6,
    bOptionMomentaryMode := GVL.bGripperScrewerOption7,
    lrPackageTurnoversToFullScrewed := lrGripperScrewerTurnoversToFullScrewed,
    lrPackageThreadPitch := lrGripperScrewerThreadPitch,
    lrPackageThreadTimes := lrGripperScrewerThreadTimes,
    lrHeightReadyPosition := lrGripperScrewerReadyPosition,
    lrHeightPushingPosition := lrGripperScrewerPushingCapPosition,
    lrHeightEndScrewingPosition := lrGripperScrewerScrewingCapPosition,
    lrHeightActualPosition := aGripperScrewer1LiftAxisRef.NcToPlc.ActPos,
    lrSpringHeightCV := IlrGripperScrewer1HeightCV,
    rActualMotor1Temperature := IrGripperScrewer1ActualMotorTemperature,
    iHeightSetTorque := 2000,
    iScrewTightTime := nGripperScrewerTightTime,
    lrScrewer1ActualTorque := aGripperScrewer1AxisRef.NcToPlc.ActTorque,
    lrHeightAcceleration := (*lrGripperScrewerLiftAcceleration*) 10000,
    lrHeightDeceleration := (*lrGripperScrewerLiftDeceleration*) 10000,
    lrHeightSpeed := (*lrGripperScrewerLiftVelocity*)700,
    lrScrewer1ActualPosition := aGripperScrewer1AxisRef.NcToPlc.ActPos,
    lrScrewerAcceleration := (100/60)*360 (*obr na st.*)(*Na stałe w bloczku*),
    lrScrewerDeceleration := 15000(*Na stałe w bloczku*),
    lrScrewerSpeed := (GVL.lrGripperScrewerVelocity/60)*360 (*obr na st.*),
    lrScrewer1PosDiff := GVL.aGripperScrewer1AxisRef.NcToPlc.PosDiff,
    lrFindigScrewDegree := lrGripperScrewerFindingScrewDegree,
    bManualMovement := bManualMode,
    lrManualOverride := VIS.lrGripperScrewerManualOverride,
    lrMaxHeightPosition := 365,
    lrMinHeightPosition := VIS.lrGripperScrewerCatchHeightCV(*+10*),
    lrMaxScrewerSpeed := 4000,
    iStationIndex := 56,
    sStationName := "Zakręcarka szczękowa 1",
    bManualHeightUp := VIS.bGripperScrewerLiftManualHeightUp,
    bManualHeightDown := VIS.bGripperScrewerLiftManualHeightDown,
    bManualScrew1Clockwise := VIS.bGripperScrewer1ManualRight,
    bManualScrew1CClockwise := VIS.bGripperScrewer1ManualLeft,
    bManualScrew2Clockwise := btemp,
    bManualScrew2CClockwise := btemp,
    bManualGripper1 := VIS.bGripperScrewer1ManualCatch,
    bManualGripper2 := btemp,
    HeightAxisRef := aGripperScrewer1LiftAxisRef,
    Screwing1AxisRef := aGripperScrewer1AxisRef,
    Screwing2AxisRef := atemp1,
    bFindScrewAdjustSensorHeight := bGripperScrewerFindScrewAdjust,
    bAdjustingTorque := bGripperScrewer1AdjustTorqueDialog,
    lrAdjustingSetTorque := VIS.lrGripperScrewer1AdjustingSetTorque,
    eRunningState => eGripperScrewer1RunningState,
    bError => GripperScrewer1Error.bError,
    udiErrorID => GripperScrewer1Error.nErrorCode,
    sErrorDescription => GripperScrewer1Error.sErrorString,
    sErrorDescription2 => GripperScrewer1Error.sErrorString2,
    sErrorStationName => GripperScrewer1Error.sStationName,
    udiStationID => GripperScrewer1Error.udiStationID,
    bGripper1Actuator => QbGripperScrewer1Actuator,
    uiScrewing1TorqueControl => QnGripperScrewer1TorqueLimit,
    rScrewing1ProportionalGain => QnGripperScrewer1ProportionalGain,
    lrScrewer1TorqueCV => VIS.lrGripperScrewer1TorqueCV,
    AsToolDescription => VIS.AsGripperScrewerTool); // FB_2GripperScrewers
eGripperScrewer1State := fb2GripperScrewer1.eState;

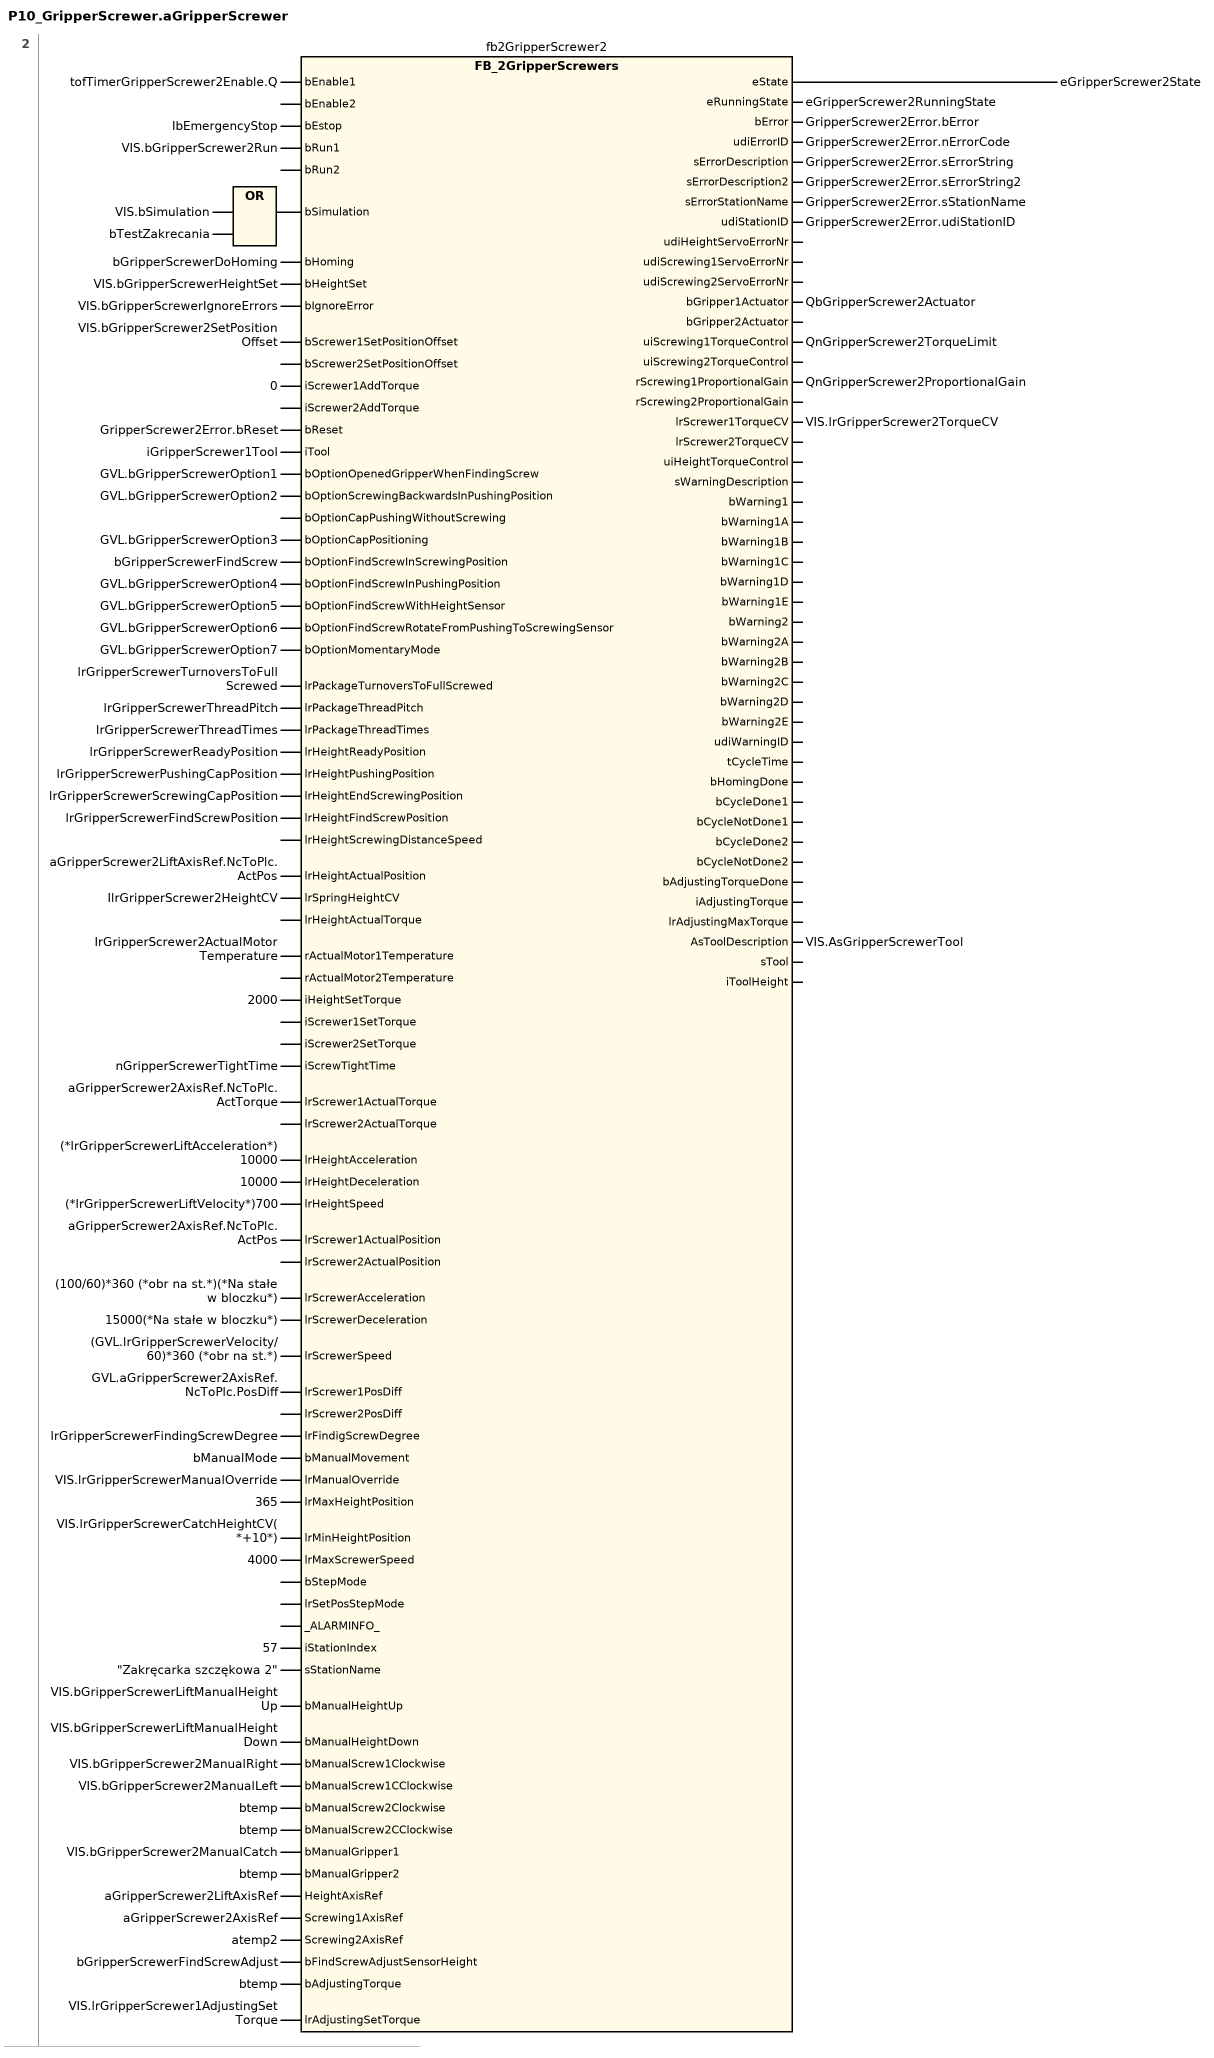
// NETWORK 2
fb2GripperScrewer2(
    bEnable1 := tofTimerGripperScrewer2Enable.Q,
    bEstop := IbEmergencyStop,
    bRun1 := VIS.bGripperScrewer2Run,
    bSimulation := VIS.bSimulation OR bTestZakrecania,
    bHoming := bGripperScrewerDoHoming,
    bHeightSet := VIS.bGripperScrewerHeightSet,
    bIgnoreError := VIS.bGripperScrewerIgnoreErrors,
    bScrewer1SetPositionOffset := VIS.bGripperScrewer2SetPositionOffset,
    iScrewer1AddTorque := 0,
    bReset := GripperScrewer2Error.bReset,
    iTool := iGripperScrewer1Tool,
    bOptionOpenedGripperWhenFindingScrew := GVL.bGripperScrewerOption1,
    bOptionScrewingBackwardsInPushingPosition := GVL.bGripperScrewerOption2,
    bOptionCapPositioning := GVL.bGripperScrewerOption3,
    bOptionFindScrewInScrewingPosition := bGripperScrewerFindScrew,
    bOptionFindScrewInPushingPosition := GVL.bGripperScrewerOption4,
    bOptionFindScrewWithHeightSensor := GVL.bGripperScrewerOption5,
    bOptionFindScrewRotateFromPushingToScrewingSensor := GVL.bGripperScrewerOption6,
    bOptionMomentaryMode := GVL.bGripperScrewerOption7,
    lrPackageTurnoversToFullScrewed := lrGripperScrewerTurnoversToFullScrewed,
    lrPackageThreadPitch := lrGripperScrewerThreadPitch,
    lrPackageThreadTimes := lrGripperScrewerThreadTimes,
    lrHeightReadyPosition := lrGripperScrewerReadyPosition,
    lrHeightPushingPosition := lrGripperScrewerPushingCapPosition,
    lrHeightEndScrewingPosition := lrGripperScrewerScrewingCapPosition,
    lrHeightFindScrewPosition := lrGripperScrewerFindScrewPosition,
    lrHeightActualPosition := aGripperScrewer2LiftAxisRef.NcToPlc.ActPos,
    lrSpringHeightCV := IlrGripperScrewer2HeightCV,
    rActualMotor1Temperature := IrGripperScrewer2ActualMotorTemperature,
    iHeightSetTorque := 2000,
    iScrewTightTime := nGripperScrewerTightTime,
    lrScrewer1ActualTorque := aGripperScrewer2AxisRef.NcToPlc.ActTorque,
    lrHeightAcceleration := (*lrGripperScrewerLiftAcceleration*) 10000,
    lrHeightDeceleration := 10000,
    lrHeightSpeed := (*lrGripperScrewerLiftVelocity*)700,
    lrScrewer1ActualPosition := aGripperScrewer2AxisRef.NcToPlc.ActPos,
    lrScrewerAcceleration := (100/60)*360 (*obr na st.*)(*Na stałe w bloczku*),
    lrScrewerDeceleration := 15000(*Na stałe w bloczku*),
    lrScrewerSpeed := (GVL.lrGripperScrewerVelocity/60)*360 (*obr na st.*),
    lrScrewer1PosDiff := GVL.aGripperScrewer2AxisRef.NcToPlc.PosDiff,
    lrFindigScrewDegree := lrGripperScrewerFindingScrewDegree,
    bManualMovement := bManualMode,
    lrManualOverride := VIS.lrGripperScrewerManualOverride,
    lrMaxHeightPosition := 365,
    lrMinHeightPosition := VIS.lrGripperScrewerCatchHeightCV(*+10*),
    lrMaxScrewerSpeed := 4000,
    iStationIndex := 57,
    sStationName := "Zakręcarka szczękowa 2",
    bManualHeightUp := VIS.bGripperScrewerLiftManualHeightUp,
    bManualHeightDown := VIS.bGripperScrewerLiftManualHeightDown,
    bManualScrew1Clockwise := VIS.bGripperScrewer2ManualRight,
    bManualScrew1CClockwise := VIS.bGripperScrewer2ManualLeft,
    bManualScrew2Clockwise := btemp,
    bManualScrew2CClockwise := btemp,
    bManualGripper1 := VIS.bGripperScrewer2ManualCatch,
    bManualGripper2 := btemp,
    HeightAxisRef := aGripperScrewer2LiftAxisRef,
    Screwing1AxisRef := aGripperScrewer2AxisRef,
    Screwing2AxisRef := atemp2,
    bFindScrewAdjustSensorHeight := bGripperScrewerFindScrewAdjust,
    bAdjustingTorque := btemp,
    lrAdjustingSetTorque := VIS.lrGripperScrewer1AdjustingSetTorque,
    eRunningState => eGripperScrewer2RunningState,
    bError => GripperScrewer2Error.bError,
    udiErrorID => GripperScrewer2Error.nErrorCode,
    sErrorDescription => GripperScrewer2Error.sErrorString,
    sErrorDescription2 => GripperScrewer2Error.sErrorString2,
    sErrorStationName => GripperScrewer2Error.sStationName,
    udiStationID => GripperScrewer2Error.udiStationID,
    bGripper1Actuator => QbGripperScrewer2Actuator,
    uiScrewing1TorqueControl => QnGripperScrewer2TorqueLimit,
    rScrewing1ProportionalGain => QnGripperScrewer2ProportionalGain,
    lrScrewer1TorqueCV => VIS.lrGripperScrewer2TorqueCV,
    AsToolDescription => VIS.AsGripperScrewerTool); // FB_2GripperScrewers
eGripperScrewer2State := fb2GripperScrewer2.eState;
END_ACTION

ACTION aGripperScrewerChartHMI:
(*Wykres zakręcarki szczękowej*)

//Zakręcarka numer 1
rtStartGripper1Screwing(CLK:=VIS.bGripperScrewer1Run, Q=>);

IF rtStartGripper1Screwing.Q THEN (*Przy starcie zarkęcania, zapamiętywanie pozycji poczatkowej*)
	lrGripperScrewer1AxisStartPosition 								:= aGripperScrewer1AxisRef.NcToPlc.ActPos;
END_IF

 fbGripperScrewer1Chart(
	bWrite															:= VIS.bGripperScrewer1Run, 
	nCycleTime														:= 5, 
	lrData1															:= VIS.lrGripperScrewer1LiftActPos, 
	lrData2															:= aGripperScrewer1AxisRef.NcToPlc.ActPos - lrGripperScrewer1AxisStartPosition,  (*Odjęcie pozycji poczatkowej*) 
//	lrData2B														:= INT_TO_LREAL(LREAL_TO_INT( LREAL_TO_REAL((aGripperScrewer1AxisRef.NcToPlc.ActTorque*1.5)/100)*100.0)) / 100.0,
	lrData2B														:= aGripperScrewer1AxisRef.NcToPlc.ActVelo/1000.0,	//(GVL.lrGripperScrewerVelocity/60)*360
	bData3															:= QbGripperScrewer1Actuator, 
	bData4															:= FALSE,
	bData5															:= FALSE,
	bData2B_ON														:= TRUE,
	AsData															=> VIS.AsChartGripperScrewer1 );
	
 fbGripperScrewer1StChart(
	bWrite															:= VIS.bGripperScrewer1Run, 
	udiCycleTime													:= TIME_TO_UDINT(fb2GripperScrewer1.tCycleTime),
	lrAiData0														:= VIS.lrGripperScrewer1LiftActPos, 
	lrAiData1														:= (aGripperScrewer1AxisRef.NcToPlc.ActPos - lrGripperScrewer1AxisStartPosition)/360.0,  (*Odjęcie pozycji poczatkowej*) 
	lrAiData2														:= aGripperScrewer1AxisRef.NcToPlc.ActVelo/100.0,	//(GVL.lrGripperScrewerVelocity/60)*360
	lrAiData3														:= BOOL_TO_LREAL(QbGripperScrewer1Actuator), 
	lrAiData4														:= IlrGripperScrewer1HeightCV, 
	AiData															=> VIS.AStChartGripperScrewer1[0] );

//Zakręcarka numer 2
rtStartGripper2Screwing(CLK:=VIS.bGripperScrewer2Run, Q=>);

IF rtStartGripper2Screwing.Q THEN (*Przy starcie zarkęcania, zapamiętywanie pozycji poczatkowej*)
	lrGripperScrewer2AxisStartPosition 								:= aGripperScrewer2AxisRef.NcToPlc.ActPos;
END_IF

 fbGripperScrewer2Chart(
	bWrite															:= VIS.bGripperScrewer2Run, 
	nCycleTime														:= 5, 
	lrData1															:= VIS.lrGripperScrewer2LiftActPos, 
	lrData2															:= aGripperScrewer2AxisRef.NcToPlc.ActPos - lrGripperScrewer2AxisStartPosition,  (*Odjęcie pozycji poczatkowej*) 
//	lrData2B														:= INT_TO_LREAL(LREAL_TO_INT( LREAL_TO_REAL((aGripperScrewer2AxisRef.NcToPlc.ActTorque*1.5)/100)*100.0)) / 100.0,
	lrData2B														:= aGripperScrewer2AxisRef.NcToPlc.ActVelo/1000.0,
	bData3															:= QbGripperScrewer2Actuator, 
	bData4															:= FALSE,
	bData5															:= FALSE,
	bData2B_ON														:= TRUE,
	AsData															=> VIS.AsChartGripperScrewer2 );

 fbGripperScrewer2StChart(
	bWrite															:= VIS.bGripperScrewer2Run, 
	udiCycleTime													:= TIME_TO_UDINT(fb2GripperScrewer2.tCycleTime),
	lrAiData0														:= VIS.lrGripperScrewer2LiftActPos, 
	lrAiData1														:= (aGripperScrewer2AxisRef.NcToPlc.ActPos - lrGripperScrewer2AxisStartPosition)/360.0,  (*Odjęcie pozycji poczatkowej*) 
	lrAiData2														:= VIS.lrGripperScrewer2TorqueCV,//aGripperScrewer2AxisRef.NcToPlc.ActVelo/100.0,	//(GVL.lrGripperScrewerVelocity/60)*360
	lrAiData3														:= BOOL_TO_LREAL(QbGripperScrewer2Actuator), 
	lrAiData4														:= IlrGripperScrewer2HeightCV, 
	AiData															=> VIS.AStChartGripperScrewer2[0] );
END_ACTION

ACTION aGripperScrewerDialogBox:

VIS.bGripperScrewer1AdjustTorque;			//Włączenie szukania
VIS.lrGripperScrewer1AdjustingSetTorque;		//Zadany moment
fb2GripperScrewer1.bAdjustingTorqueDone; 		//Wykonano badanie
fb2GripperScrewer1.iAdjustingTorque; 			//Wynik badania

	(*Informacja o opcji szukania momentu otwierania*)		
	IF VIS.bGripperScrewer1AdjustTorque THEN
		
		CASE nGripperScrewer1AdjustingDialog OF
			
			0: //Zerowanie
				nGripperScrewer1AdjustingDialog								:= 1;
				
			1: //Czy rozpocząć?
				VIS.nDialogBoxType											:= 3;
				VIS.bDialogBoxText											:= 'Rozpocznij szukanie momentu otwierania, czy zjechałeś stacją na wysokość zakręcania?';
				VIS.bDialogBoxText2											:= '';
				VIS.sDialogBoxPicture										:= '1';
				VIS.bDialogBoxOn											:= TRUE;
				
				IF VIS.bDialogBoxAck THEN
					VIS.bDialogBoxAck										:= FALSE;
					nGripperScrewer1AdjustingDialog							:= 2;
				END_IF
				
				IF VIS.bDialogBoxCancelAck THEN
					nGripperScrewer1AdjustingDialog							:= 1;
					P00_Visualization.aResetDialog();
					VIS.bGripperScrewer1AdjustTorque						:= FALSE;	
				END_IF
				
				
			2: //Trwa..
				bGripperScrewer1AdjustTorqueDialog							:= TRUE; 	// Włączenie szukania
				VIS.nDialogBoxType											:= 2;
				VIS.bDialogBoxText											:= 'Trwa szukanie momentu otwierania [Nm]';
				VIS.bDialogBoxText2											:= REAL_TO_STRING(LREAL_TO_REAL(fb2GripperScrewer1.lrAdjustingMaxTorque));
				VIS.sDialogBoxPicture										:= '1';
				VIS.bDialogBoxOn											:= TRUE;
				
				IF fb2GripperScrewer1.bAdjustingTorqueDone THEN
					nGripperScrewer1AdjustingDialog							:= 3;
					nTstcount												:= nTstcount+1;
				END_IF
				
				IF VIS.bDialogBoxCancelAck THEN
					nGripperScrewer1AdjustingDialog							:= 0;
					P00_Visualization.aResetDialog();
					VIS.bGripperScrewer1AdjustTorque						:= FALSE;
					bGripperScrewer1AdjustTorqueDialog 						:= FALSE;
				END_IF
				
				
			3: //Ustawiony moment
				VIS.nDialogBoxType											:= 1;		// Przycisk TAK
				VIS.bDialogBoxText											:= 'Nastawa momentu zakręcania [%] została ustawiona na:';
				VIS.bDialogBoxText2											:= INT_TO_STRING(fb2GripperScrewer1.iAdjustingTorque);
				VIS.sDialogBoxPicture										:= '1';
				VIS.bDialogBoxOn											:= TRUE;
				VIS.lrGripperScrewingTightTorqueShow						:= fb2GripperScrewer1.iAdjustingTorque;
				
				IF VIS.bDialogBoxAck THEN
					VIS.bDialogBoxAck 										:= FALSE;
					nGripperScrewer1AdjustingDialog							:= 0;
					VIS.bGripperScrewer1AdjustTorque						:= FALSE;
					bGripperScrewer1AdjustTorqueDialog						:= FALSE;
					P00_Visualization.aResetDialog();
				END_IF
				
		END_CASE
	END_IF
	(*Koniec Informacja o opcji szukania momentu otwierania*)
	///
END_ACTION

ACTION aGripperScrewerEnable:
(*Opoznienie wyłączanie enabla dozownikow*)
(*Nie zdarzy wyjśc z Disabled podczas zmiany recepptury*)
tofTimerGripperScrewer1Enable(IN:=bGripperScrewer1Enable (*AND NOT bChangeover*), PT:=T#1S);
tofTimerGripperScrewer2Enable(IN:=bGripperScrewer2Enable (*AND NOT bChangeover*), PT:=T#1S);


(*Wyłączanie dozowników parami*)
bGripperScrewer1Enable				:= bGripperScrewer1Enable AND bGripperScrewer2Enable;
bGripperScrewer2Enable 				:= bGripperScrewer1Enable AND bGripperScrewer2Enable;

(*Ustawianie zmiennych wizualizacyjnych*)
rtbGripperScrewer12EnableShow		(CLK:=VIS.bGripperScrewer1EnableShow OR VIS.bGripperScrewer2EnableShow,Q=>);
IF rtbGripperScrewer12EnableShow.Q THEN
	VIS.bGripperScrewer1EnableShow  := TRUE;
	VIS.bGripperScrewer2EnableShow	:= TRUE;	
END_IF
ftbGripperScrewer12EnableShow		(CLK:=VIS.bGripperScrewer1EnableShow AND VIS.bGripperScrewer2EnableShow,Q=>);
IF ftbGripperScrewer12EnableShow.Q THEN
	VIS.bGripperScrewer1EnableShow  := FALSE;
	VIS.bGripperScrewer2EnableShow 	:= FALSE;	
END_IF
END_ACTION

ACTION aGripperScrewerNew:
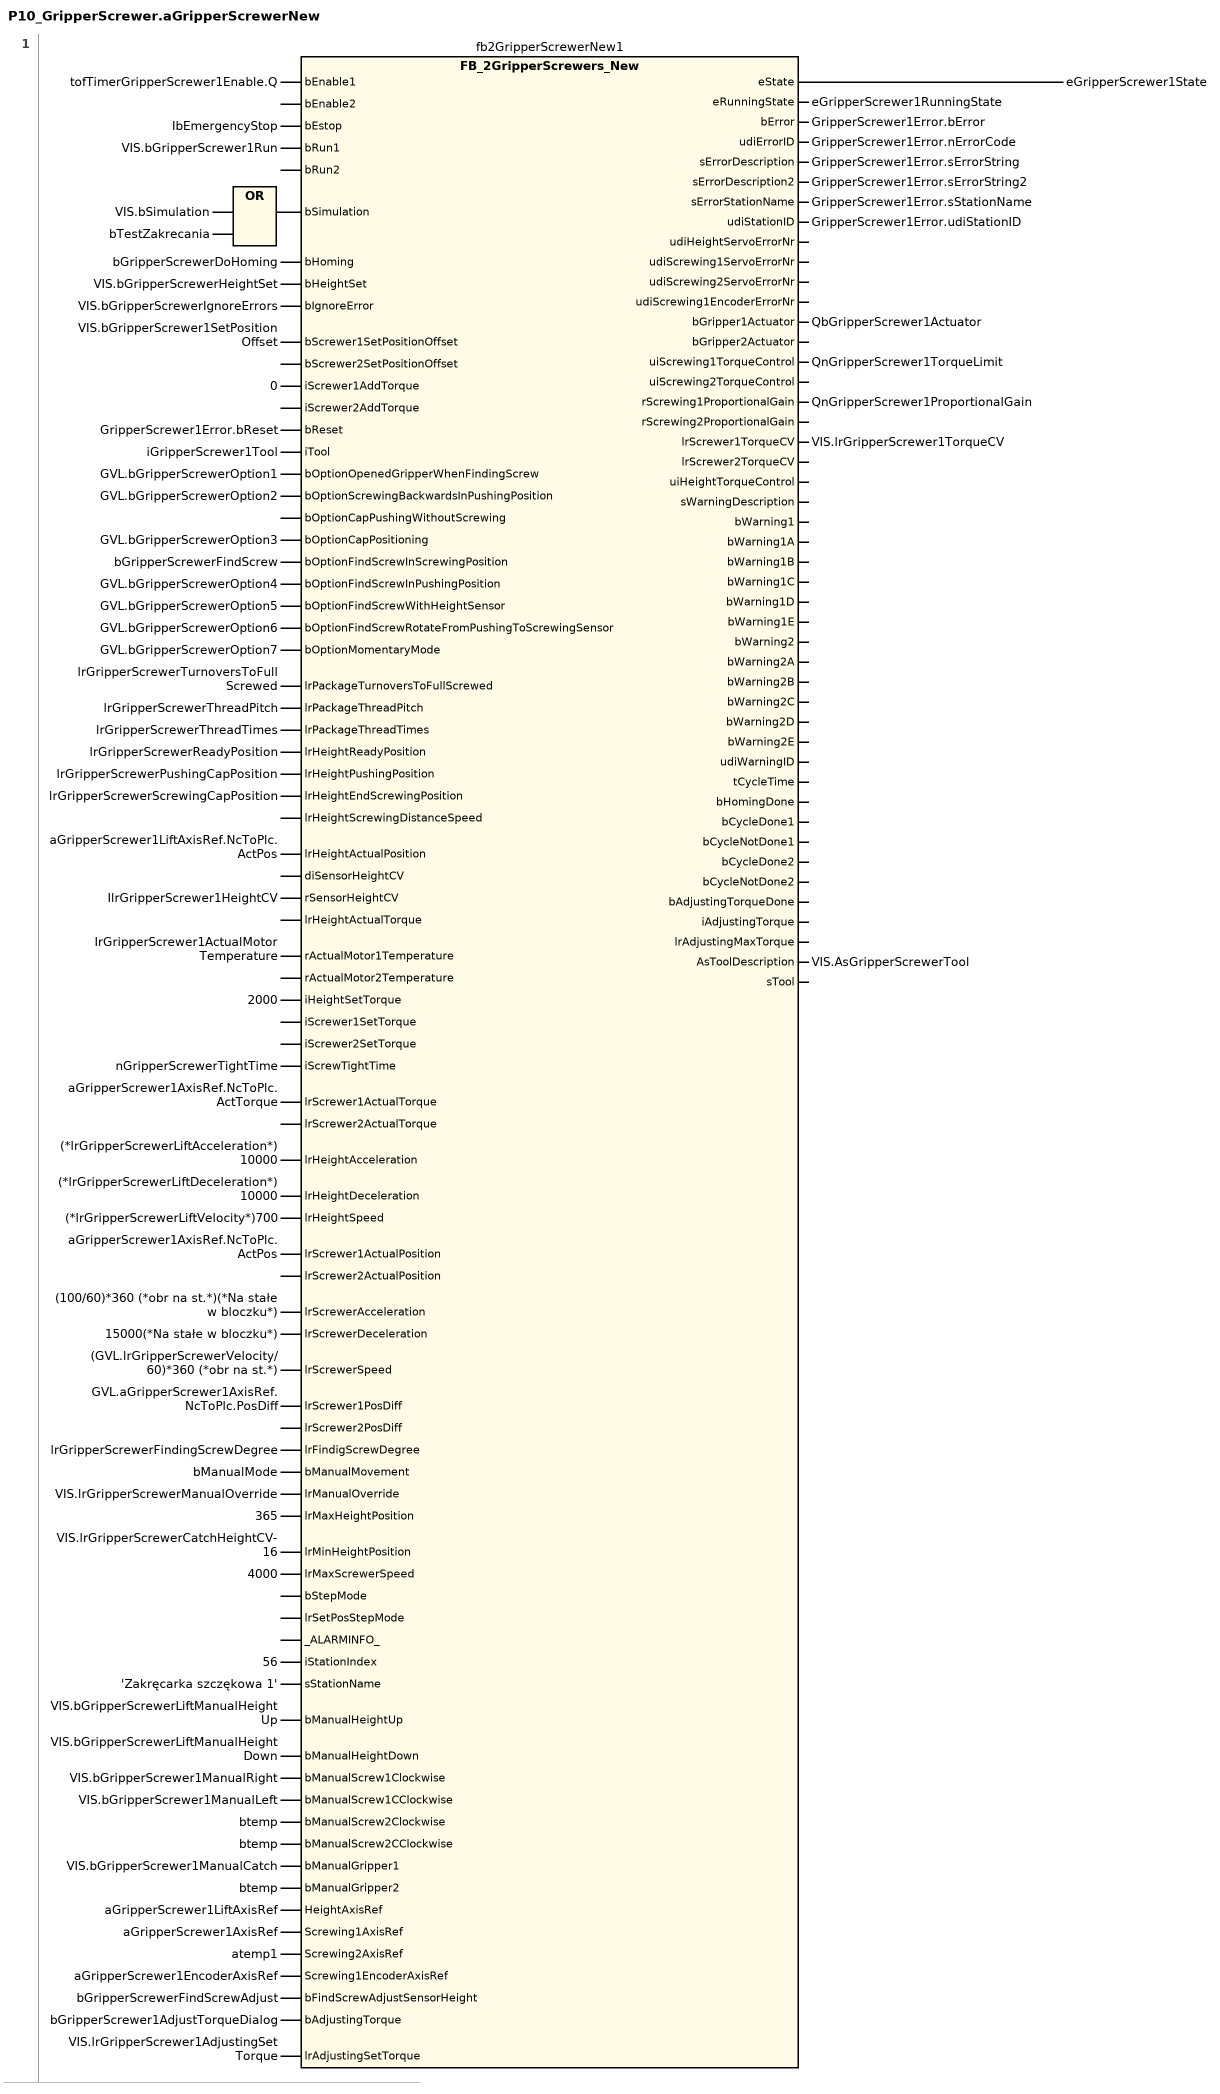
// NETWORK 1
fb2GripperScrewerNew1(
    bEnable1 := tofTimerGripperScrewer1Enable.Q,
    bEstop := IbEmergencyStop,
    bRun1 := VIS.bGripperScrewer1Run,
    bSimulation := VIS.bSimulation OR bTestZakrecania,
    bHoming := bGripperScrewerDoHoming,
    bHeightSet := VIS.bGripperScrewerHeightSet,
    bIgnoreError := VIS.bGripperScrewerIgnoreErrors,
    bScrewer1SetPositionOffset := VIS.bGripperScrewer1SetPositionOffset,
    iScrewer1AddTorque := 0,
    bReset := GripperScrewer1Error.bReset,
    iTool := iGripperScrewer1Tool,
    bOptionOpenedGripperWhenFindingScrew := GVL.bGripperScrewerOption1,
    bOptionScrewingBackwardsInPushingPosition := GVL.bGripperScrewerOption2,
    bOptionCapPositioning := GVL.bGripperScrewerOption3,
    bOptionFindScrewInScrewingPosition := bGripperScrewerFindScrew,
    bOptionFindScrewInPushingPosition := GVL.bGripperScrewerOption4,
    bOptionFindScrewWithHeightSensor := GVL.bGripperScrewerOption5,
    bOptionFindScrewRotateFromPushingToScrewingSensor := GVL.bGripperScrewerOption6,
    bOptionMomentaryMode := GVL.bGripperScrewerOption7,
    lrPackageTurnoversToFullScrewed := lrGripperScrewerTurnoversToFullScrewed,
    lrPackageThreadPitch := lrGripperScrewerThreadPitch,
    lrPackageThreadTimes := lrGripperScrewerThreadTimes,
    lrHeightReadyPosition := lrGripperScrewerReadyPosition,
    lrHeightPushingPosition := lrGripperScrewerPushingCapPosition,
    lrHeightEndScrewingPosition := lrGripperScrewerScrewingCapPosition,
    lrHeightActualPosition := aGripperScrewer1LiftAxisRef.NcToPlc.ActPos,
    rSensorHeightCV := IlrGripperScrewer1HeightCV,
    rActualMotor1Temperature := IrGripperScrewer1ActualMotorTemperature,
    iHeightSetTorque := 2000,
    iScrewTightTime := nGripperScrewerTightTime,
    lrScrewer1ActualTorque := aGripperScrewer1AxisRef.NcToPlc.ActTorque,
    lrHeightAcceleration := (*lrGripperScrewerLiftAcceleration*) 10000,
    lrHeightDeceleration := (*lrGripperScrewerLiftDeceleration*) 10000,
    lrHeightSpeed := (*lrGripperScrewerLiftVelocity*)700,
    lrScrewer1ActualPosition := aGripperScrewer1AxisRef.NcToPlc.ActPos,
    lrScrewerAcceleration := (100/60)*360 (*obr na st.*)(*Na stałe w bloczku*),
    lrScrewerDeceleration := 15000(*Na stałe w bloczku*),
    lrScrewerSpeed := (GVL.lrGripperScrewerVelocity/60)*360 (*obr na st.*),
    lrScrewer1PosDiff := GVL.aGripperScrewer1AxisRef.NcToPlc.PosDiff,
    lrFindigScrewDegree := lrGripperScrewerFindingScrewDegree,
    bManualMovement := bManualMode,
    lrManualOverride := VIS.lrGripperScrewerManualOverride,
    lrMaxHeightPosition := 365,
    lrMinHeightPosition := VIS.lrGripperScrewerCatchHeightCV-16,
    lrMaxScrewerSpeed := 4000,
    iStationIndex := 56,
    sStationName := 'Zakręcarka szczękowa 1',
    bManualHeightUp := VIS.bGripperScrewerLiftManualHeightUp,
    bManualHeightDown := VIS.bGripperScrewerLiftManualHeightDown,
    bManualScrew1Clockwise := VIS.bGripperScrewer1ManualRight,
    bManualScrew1CClockwise := VIS.bGripperScrewer1ManualLeft,
    bManualScrew2Clockwise := btemp,
    bManualScrew2CClockwise := btemp,
    bManualGripper1 := VIS.bGripperScrewer1ManualCatch,
    bManualGripper2 := btemp,
    HeightAxisRef := aGripperScrewer1LiftAxisRef,
    Screwing1AxisRef := aGripperScrewer1AxisRef,
    Screwing2AxisRef := atemp1,
    Screwing1EncoderAxisRef := aGripperScrewer1EncoderAxisRef,
    bFindScrewAdjustSensorHeight := bGripperScrewerFindScrewAdjust,
    bAdjustingTorque := bGripperScrewer1AdjustTorqueDialog,
    lrAdjustingSetTorque := VIS.lrGripperScrewer1AdjustingSetTorque,
    eRunningState => eGripperScrewer1RunningState,
    bError => GripperScrewer1Error.bError,
    udiErrorID => GripperScrewer1Error.nErrorCode,
    sErrorDescription => GripperScrewer1Error.sErrorString,
    sErrorDescription2 => GripperScrewer1Error.sErrorString2,
    sErrorStationName => GripperScrewer1Error.sStationName,
    udiStationID => GripperScrewer1Error.udiStationID,
    bGripper1Actuator => QbGripperScrewer1Actuator,
    uiScrewing1TorqueControl => QnGripperScrewer1TorqueLimit,
    rScrewing1ProportionalGain => QnGripperScrewer1ProportionalGain,
    lrScrewer1TorqueCV => VIS.lrGripperScrewer1TorqueCV,
    AsToolDescription => VIS.AsGripperScrewerTool); // FB_2GripperScrewers_New
eGripperScrewer1State := fb2GripperScrewerNew1.eState;

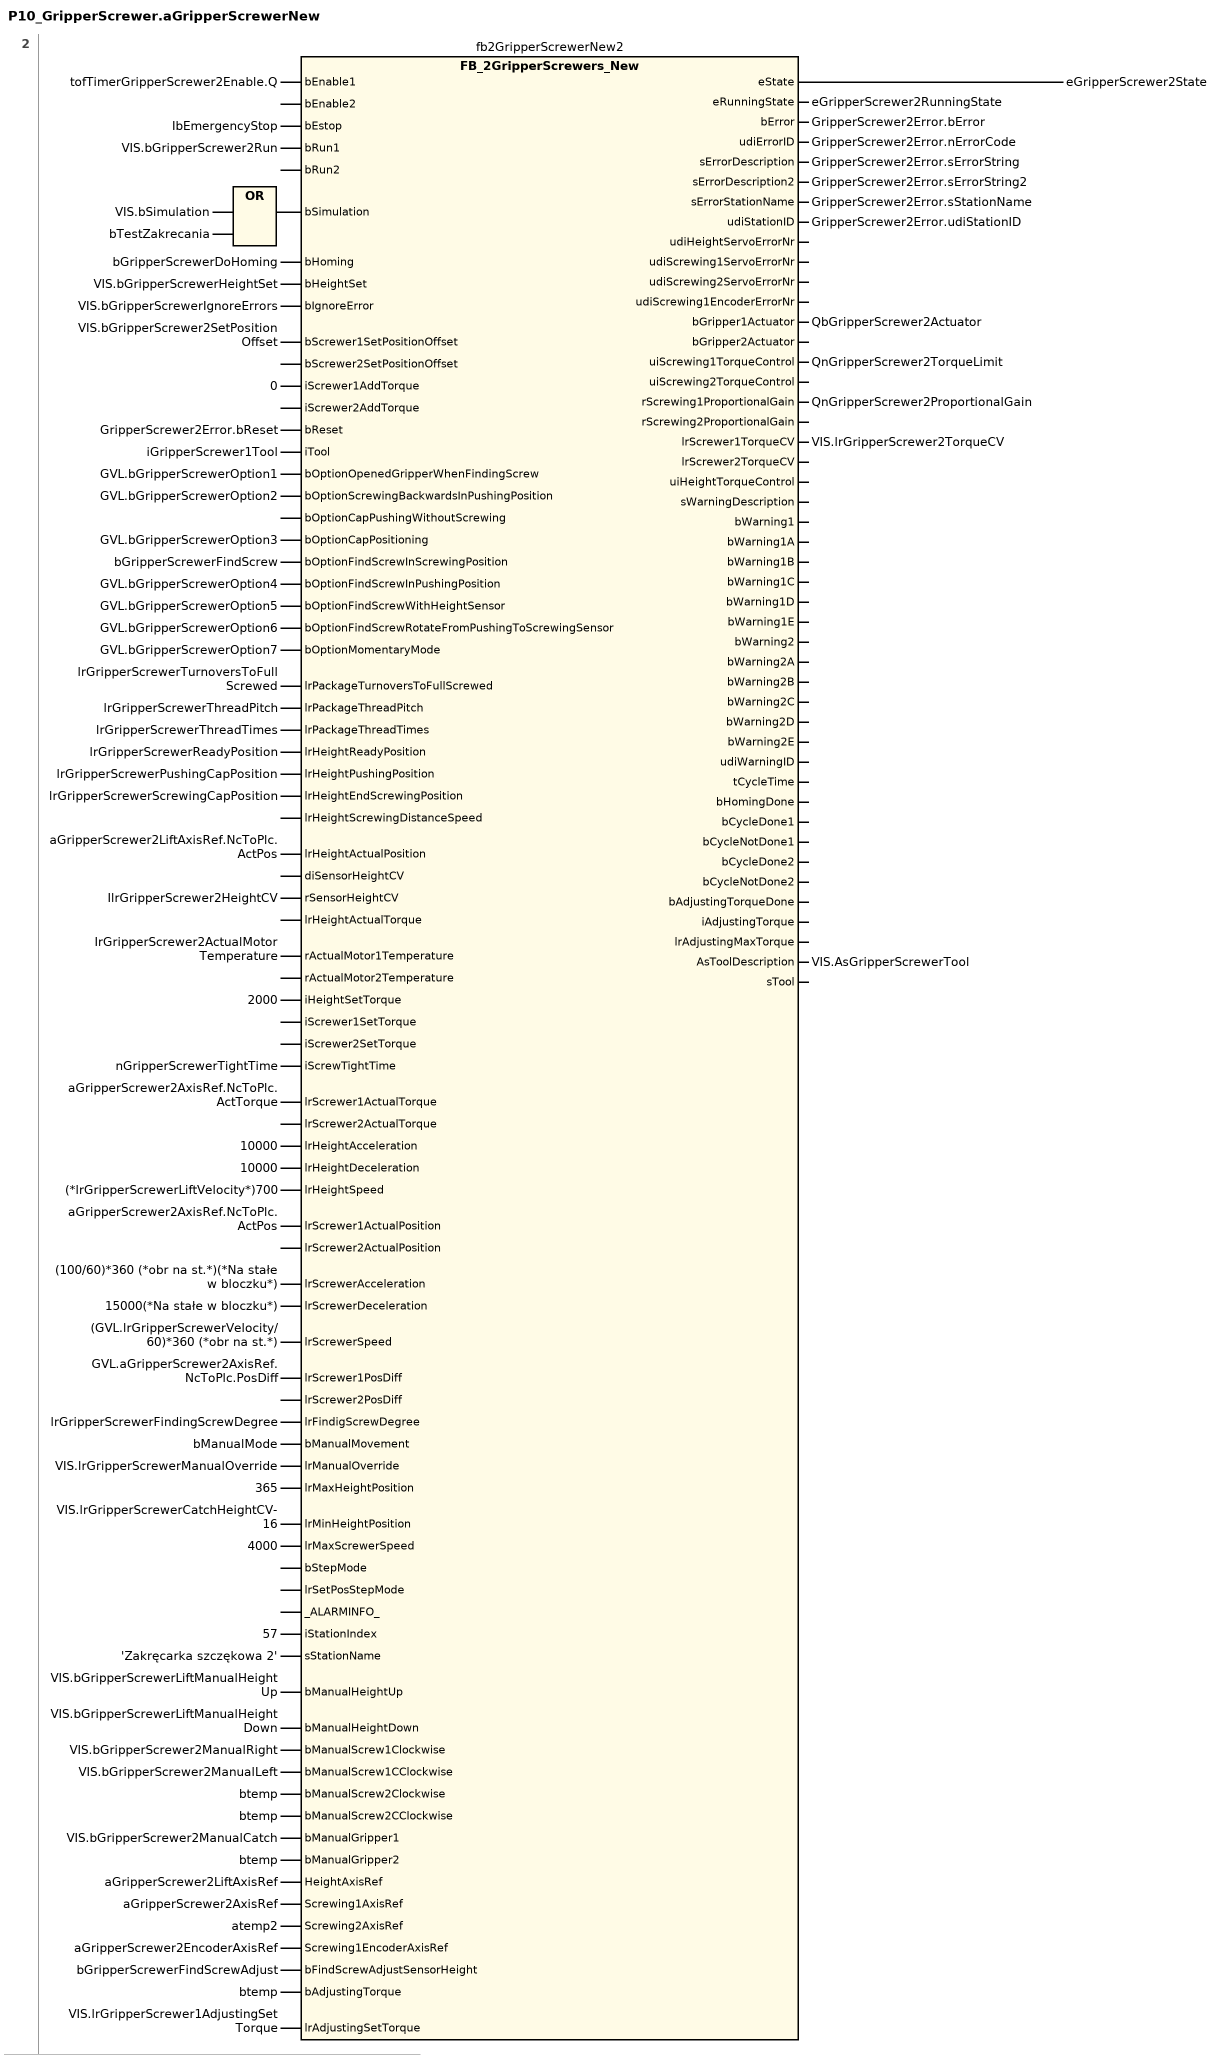
// NETWORK 2
fb2GripperScrewerNew2(
    bEnable1 := tofTimerGripperScrewer2Enable.Q,
    bEstop := IbEmergencyStop,
    bRun1 := VIS.bGripperScrewer2Run,
    bSimulation := VIS.bSimulation OR bTestZakrecania,
    bHoming := bGripperScrewerDoHoming,
    bHeightSet := VIS.bGripperScrewerHeightSet,
    bIgnoreError := VIS.bGripperScrewerIgnoreErrors,
    bScrewer1SetPositionOffset := VIS.bGripperScrewer2SetPositionOffset,
    iScrewer1AddTorque := 0,
    bReset := GripperScrewer2Error.bReset,
    iTool := iGripperScrewer1Tool,
    bOptionOpenedGripperWhenFindingScrew := GVL.bGripperScrewerOption1,
    bOptionScrewingBackwardsInPushingPosition := GVL.bGripperScrewerOption2,
    bOptionCapPositioning := GVL.bGripperScrewerOption3,
    bOptionFindScrewInScrewingPosition := bGripperScrewerFindScrew,
    bOptionFindScrewInPushingPosition := GVL.bGripperScrewerOption4,
    bOptionFindScrewWithHeightSensor := GVL.bGripperScrewerOption5,
    bOptionFindScrewRotateFromPushingToScrewingSensor := GVL.bGripperScrewerOption6,
    bOptionMomentaryMode := GVL.bGripperScrewerOption7,
    lrPackageTurnoversToFullScrewed := lrGripperScrewerTurnoversToFullScrewed,
    lrPackageThreadPitch := lrGripperScrewerThreadPitch,
    lrPackageThreadTimes := lrGripperScrewerThreadTimes,
    lrHeightReadyPosition := lrGripperScrewerReadyPosition,
    lrHeightPushingPosition := lrGripperScrewerPushingCapPosition,
    lrHeightEndScrewingPosition := lrGripperScrewerScrewingCapPosition,
    lrHeightActualPosition := aGripperScrewer2LiftAxisRef.NcToPlc.ActPos,
    rSensorHeightCV := IlrGripperScrewer2HeightCV,
    rActualMotor1Temperature := IrGripperScrewer2ActualMotorTemperature,
    iHeightSetTorque := 2000,
    iScrewTightTime := nGripperScrewerTightTime,
    lrScrewer1ActualTorque := aGripperScrewer2AxisRef.NcToPlc.ActTorque,
    lrHeightAcceleration := 10000,
    lrHeightDeceleration := 10000,
    lrHeightSpeed := (*lrGripperScrewerLiftVelocity*)700,
    lrScrewer1ActualPosition := aGripperScrewer2AxisRef.NcToPlc.ActPos,
    lrScrewerAcceleration := (100/60)*360 (*obr na st.*)(*Na stałe w bloczku*),
    lrScrewerDeceleration := 15000(*Na stałe w bloczku*),
    lrScrewerSpeed := (GVL.lrGripperScrewerVelocity/60)*360 (*obr na st.*),
    lrScrewer1PosDiff := GVL.aGripperScrewer2AxisRef.NcToPlc.PosDiff,
    lrFindigScrewDegree := lrGripperScrewerFindingScrewDegree,
    bManualMovement := bManualMode,
    lrManualOverride := VIS.lrGripperScrewerManualOverride,
    lrMaxHeightPosition := 365,
    lrMinHeightPosition := VIS.lrGripperScrewerCatchHeightCV-16,
    lrMaxScrewerSpeed := 4000,
    iStationIndex := 57,
    sStationName := 'Zakręcarka szczękowa 2',
    bManualHeightUp := VIS.bGripperScrewerLiftManualHeightUp,
    bManualHeightDown := VIS.bGripperScrewerLiftManualHeightDown,
    bManualScrew1Clockwise := VIS.bGripperScrewer2ManualRight,
    bManualScrew1CClockwise := VIS.bGripperScrewer2ManualLeft,
    bManualScrew2Clockwise := btemp,
    bManualScrew2CClockwise := btemp,
    bManualGripper1 := VIS.bGripperScrewer2ManualCatch,
    bManualGripper2 := btemp,
    HeightAxisRef := aGripperScrewer2LiftAxisRef,
    Screwing1AxisRef := aGripperScrewer2AxisRef,
    Screwing2AxisRef := atemp2,
    Screwing1EncoderAxisRef := aGripperScrewer2EncoderAxisRef,
    bFindScrewAdjustSensorHeight := bGripperScrewerFindScrewAdjust,
    bAdjustingTorque := btemp,
    lrAdjustingSetTorque := VIS.lrGripperScrewer1AdjustingSetTorque,
    eRunningState => eGripperScrewer2RunningState,
    bError => GripperScrewer2Error.bError,
    udiErrorID => GripperScrewer2Error.nErrorCode,
    sErrorDescription => GripperScrewer2Error.sErrorString,
    sErrorDescription2 => GripperScrewer2Error.sErrorString2,
    sErrorStationName => GripperScrewer2Error.sStationName,
    udiStationID => GripperScrewer2Error.udiStationID,
    bGripper1Actuator => QbGripperScrewer2Actuator,
    uiScrewing1TorqueControl => QnGripperScrewer2TorqueLimit,
    rScrewing1ProportionalGain => QnGripperScrewer2ProportionalGain,
    lrScrewer1TorqueCV => VIS.lrGripperScrewer2TorqueCV,
    AsToolDescription => VIS.AsGripperScrewerTool); // FB_2GripperScrewers_New
eGripperScrewer2State := fb2GripperScrewerNew2.eState;
END_ACTION

ACTION aGripperScrewerWarnings:
//Zakręcarka 1 - przekroczenie czasu zakręcania - zmień ust.
IF fb2GripperScrewer1.bWarning1A AND NOT ScrewersWarning[0].bWarning THEN
	ScrewersWarning[0].bWarning										:= TRUE;
	ScrewersWarning[0].udiWarningCode								:= 49;
	ScrewersWarning[0].sDescription									:= 'Zakręcarka 1 | Przekroczenie czasu zakręcania - zmień ust.';
ELSIF NOT fb2GripperScrewer1.bWarning1A  AND ScrewersWarning[0].bAcknowledge THEN
	ScrewersWarning[0].bWarning										:= FALSE;
	ScrewersWarning[0].bAcknowledge									:= FALSE;
	VIS.uliWarningAcknowledge.15 									:= FALSE;
ELSIF ScrewersWarning[0].bAcknowledge THEN
	ScrewersWarning[0].bAcknowledge									:= TRUE;
END_IF

//Zakręcarka 1 - przekroczenie czasu szukania gwintu - zmień ust.
IF fb2GripperScrewer1.bWarning1B AND NOT ScrewersWarning[1].bWarning THEN
	ScrewersWarning[1].bWarning										:= TRUE;
	ScrewersWarning[1].udiWarningCode								:= 50;
	ScrewersWarning[1].sDescription									:= 'Zakręcarka 1 | Przekroczenie czasu szukania gwintu - zmień ust.';
ELSIF NOT fb2GripperScrewer1.bWarning1B  AND ScrewersWarning[1].bAcknowledge THEN
	ScrewersWarning[1].bWarning										:= FALSE;
	ScrewersWarning[1].bAcknowledge									:= FALSE;
	VIS.uliWarningAcknowledge.16 									:= FALSE;
ELSIF ScrewersWarning[1].bAcknowledge THEN
	ScrewersWarning[1].bAcknowledge									:= TRUE;
END_IF

//Zakręcarka 1 - przekroczenie laga - zmień ust.
IF fb2GripperScrewer1.bWarning1C AND NOT ScrewersWarning[2].bWarning THEN
	ScrewersWarning[2].bWarning										:= TRUE;
	ScrewersWarning[2].udiWarningCode								:= 51;
	ScrewersWarning[2].sDescription									:= 'Zakręcarka 1 | Przekroczenie poślizgu - zmień ust.';
ELSIF NOT fb2GripperScrewer1.bWarning1C  AND ScrewersWarning[2].bAcknowledge THEN
	ScrewersWarning[2].bWarning										:= FALSE;
	ScrewersWarning[2].bAcknowledge									:= FALSE;
	VIS.uliWarningAcknowledge.17 									:= FALSE;
ELSIF ScrewersWarning[2].bAcknowledge THEN
	ScrewersWarning[2].bAcknowledge									:= TRUE;
END_IF

//Zakręcarka 1 - zbyt niska pozycja przy zakrecaniu - zmień ust.
IF fb2GripperScrewer1.bWarning1D AND NOT ScrewersWarning[3].bWarning THEN
	ScrewersWarning[3].bWarning										:= TRUE;
	ScrewersWarning[3].udiWarningCode								:= 52;
	ScrewersWarning[3].sDescription									:= 'Zakręcarka 1 | Zbyt niska pozycja przy zakrecaniu - zmień ust.';
ELSIF NOT fb2GripperScrewer1.bWarning1D  AND ScrewersWarning[3].bAcknowledge THEN
	ScrewersWarning[3].bWarning										:= FALSE;
	ScrewersWarning[3].bAcknowledge									:= FALSE;
	VIS.uliWarningAcknowledge.18 									:= FALSE;
ELSIF ScrewersWarning[3].bAcknowledge THEN
	ScrewersWarning[3].bAcknowledge									:= TRUE;
END_IF

//Zakręcarka 2 - przekroczenie czasu zakręcania - zmień ust.
IF fb2GripperScrewer2.bWarning1A AND NOT ScrewersWarning[4].bWarning THEN
	ScrewersWarning[4].bWarning										:= TRUE;
	ScrewersWarning[4].udiWarningCode								:= 53;
	ScrewersWarning[4].sDescription									:= 'Zakręcarka 2 | Przekroczenie czasu zakręcania - zmień ust.';
ELSIF NOT fb2GripperScrewer2.bWarning1A  AND ScrewersWarning[4].bAcknowledge THEN
	ScrewersWarning[4].bWarning										:= FALSE;
	ScrewersWarning[4].bAcknowledge									:= FALSE;
	VIS.uliWarningAcknowledge.19 									:= FALSE;
ELSIF ScrewersWarning[4].bAcknowledge THEN
	ScrewersWarning[4].bAcknowledge									:= TRUE;
END_IF


//Zakręcarka 2 - przekroczenie czasu szukania gwintu - zmień ust.
IF fb2GripperScrewer2.bWarning1B AND NOT ScrewersWarning[5].bWarning THEN
	ScrewersWarning[5].bWarning										:= TRUE;
	ScrewersWarning[5].udiWarningCode								:= 54;
	ScrewersWarning[5].sDescription									:= 'Zakręcarka 2 | Przekroczenie czasu szukania gwintu - zmień ust.';
ELSIF NOT fb2GripperScrewer2.bWarning1B  AND ScrewersWarning[5].bAcknowledge THEN
	ScrewersWarning[5].bWarning										:= FALSE;
	ScrewersWarning[5].bAcknowledge									:= FALSE;
	VIS.uliWarningAcknowledge.20 									:= FALSE;
ELSIF ScrewersWarning[5].bAcknowledge THEN
	ScrewersWarning[5].bAcknowledge									:= TRUE;
END_IF

//Zakręcarka 2 - przekroczenie laga - zmień ust.
IF fb2GripperScrewer2.bWarning1C AND NOT ScrewersWarning[6].bWarning THEN
	ScrewersWarning[6].bWarning										:= TRUE;
	ScrewersWarning[6].udiWarningCode								:= 55;
	ScrewersWarning[6].sDescription									:= 'Zakręcarka 2 | Przekroczenie poślizgu - zmień ust.';
ELSIF NOT fb2GripperScrewer2.bWarning1C  AND ScrewersWarning[6].bAcknowledge THEN
	ScrewersWarning[6].bWarning										:= FALSE;
	ScrewersWarning[6].bAcknowledge									:= FALSE;
	VIS.uliWarningAcknowledge.21 									:= FALSE;
ELSIF ScrewersWarning[6].bAcknowledge THEN
	ScrewersWarning[6].bAcknowledge									:= TRUE;
END_IF

//Zakręcarka 2 - zbyt niska pozycja przy zakrecaniu - zmień ust.
IF fb2GripperScrewer2.bWarning1D AND NOT ScrewersWarning[7].bWarning THEN
	ScrewersWarning[7].bWarning										:= TRUE;
	ScrewersWarning[7].udiWarningCode								:= 56;
	ScrewersWarning[7].sDescription									:= 'Zakręcarka 2 | Zbyt niska pozycja przy zakrecaniu - zmień ust.';
ELSIF NOT fb2GripperScrewer2.bWarning1D  AND ScrewersWarning[7].bAcknowledge THEN
	ScrewersWarning[7].bWarning										:= FALSE;
	ScrewersWarning[7].bAcknowledge									:= FALSE;
	VIS.uliWarningAcknowledge.22 									:= FALSE;
ELSIF ScrewersWarning[7].bAcknowledge THEN
	ScrewersWarning[7].bAcknowledge									:= TRUE;
END_IF
END_ACTION

ACTION aInfo:

// Informacja o zuzytych gumach na zakręcarce

rtfb2GripperScrewer1Done (CLK:=fb2GripperScrewer1.bCycleDone1 OR  fb2GripperScrewer1.bCycleNotDone1, Q=>);
IF rtfb2GripperScrewer1Done.Q THEN
	IF NOT fb2GripperScrewer1.bWarning1A AND NOT fb2GripperScrewer1.bWarning1C THEN
		iGripperScrewer1Info1 			:= 0;
		iGripperScrewer1NoWarningInRow	:= iGripperScrewer1NoWarningInRow	+	1;
	ELSE
		iGripperScrewer1Info1 			:= iGripperScrewer1Info1 + 1;
		iGripperScrewer1NoWarningInRow	:= 0;
	END_IF	
END_IF
	
rtfb2GripperScrewer2Done (CLK:=fb2GripperScrewer2.bCycleDone1 OR  fb2GripperScrewer2.bCycleNotDone1, Q=>);
IF rtfb2GripperScrewer2Done.Q THEN
	IF NOT fb2GripperScrewer2.bWarning1A AND NOT fb2GripperScrewer2.bWarning1C THEN
		iGripperScrewer1Info1 			:= 0;
		iGripperScrewer2NoWarningInRow	:=	iGripperScrewer2NoWarningInRow	+	1;
	ELSE
		iGripperScrewer1Info1 			:= iGripperScrewer1Info1 + 1;
		iGripperScrewer2NoWarningInRow	:= 0;
	END_IF	
END_IF


IF iGripperScrewer1Info1 >3 THEN
	bGripperScrewer1ChangeRubbers := TRUE;
END_IF
IF iGripperScrewer2Info1 >3 THEN
	bGripperScrewer2ChangeRubbers := TRUE;
END_IF
tonbGripperScrewer1ChangeRubbers (IN:=bGripperScrewer1ChangeRubbers AND iGripperScrewer1Info1<3,Q=>);
IF tonbGripperScrewer1ChangeRubbers.Q THEN
	bGripperScrewer1ChangeRubbers	:=	FALSE;
END_IF
tonbGripperScrewer2ChangeRubbers (IN:=bGripperScrewer2ChangeRubbers AND iGripperScrewer2Info1<3,Q=>);
IF tonbGripperScrewer2ChangeRubbers.Q THEN
	bGripperScrewer2ChangeRubbers	:=	FALSE;
END_IF
END_ACTION

ACTION aLimits:
(*
Nazwa:			aLimits
Opis:			Zabezpieczenia
Wersja:			v1.0
Data:			2023-11-24
Autor:			DP
Urzadzenia:		
Zmiany:	
- 20231124 [DP] Aktualizacja do nowej wersji i opisów wizki
Info:
*)

(**** Limity i zabezpieczenia***)

IF 	VIS.lrBottleDragingStationStartPosition		= 0		THEN	VIS.lrBottleDragingStationStartPosition		:=	3;		END_IF;
IF 	VIS.lrBottleDragingStationEndPosition		= 0		THEN	VIS.lrBottleDragingStationEndPosition		:=	137;	END_IF;


IF VIS.lrGripperScrewer1VelocityShow < 30 THEN
	lrGripperScrewerVelocity			:=	30;
	VIS.lrGripperScrewer1VelocityShow	:=	30;
END_IF

IF VIS.lrGripperScrewerManualOverride = 0 THEN
	VIS.lrGripperScrewerManualOverride := 100;
END_IF

IF VIS.lrGripperScrewerTurnoversToFullScrewedShow < 0.1 THEN
	VIS.lrGripperScrewerTurnoversToFullScrewedShow := 0.1;
END_IF

VIS.bGripperScrewer1FindScrewShow				;// Szukania gwintu w pozycji zakręcania						
VIS.lrGripperScrewer1FindingScrewDegreeShow		;// Kąt szukania gwintu 
VIS.iGripperScrewer1ToolShow						;// Typ narzędzia (0-3), opisy w tablicy AsGripperScrewerTool	
VIS.bGripperScrewer1Option1Show					;// Otwieraj szczęki podczas szukania gwintu
VIS.bGripperScrewer1Option2Show					;// Obrót do tyłu w pozycji dociskania
VIS.bGripperScrewer1Option3Show					;// Dodatkowy ruch chwytakiem przed zakręceniem 
VIS.bGripperScrewer1Option4Show					;// Szukanie gwintu w pozycji dociskania
VIS.bGripperScrewer1Option5Show					;// Szukanie gwintu z czujnikiem wysokości
VIS.bGripperScrewer1Option6Show					;// Obrót podczas przejścia z pozycji docisku do zakręcania podczas szukania gwintu
VIS.bGripperScrewer1Option7Show					;// Rezerwa


(****Opcja 1*****)
IF NOT VIS.bGripperScrewer1FindScrewShow AND NOT VIS.bGripperScrewer1Option4Show THEN
	VIS.bGripperScrewer1Option1Show 	:= FALSE; 	// Otwieraj szczęki podczas szukania gwintu
END_IF

(****Opcja 2*****)
IF VIS.lrGripperScrewerPushingCapPositionShow	= VIS.lrGripperScrewerScrewingCapPositionShow	OR 
	lrGripperScrewerPushingCapPosition 			= lrGripperScrewerScrewingCapPosition OR  
	VIS.bGripperScrewer1Option5Show
THEN
	VIS.bGripperScrewer1Option2Show;
	//VIS.bGripperScrewer1Option2Show := FALSE; // Obrót do tyłu w pozycji dociskania
END_IF

(****Opcja 3*****)
IF fb2GripperScrewer2.sTool = 'ksztalkowa/do kulek' OR fb2GripperScrewer2.sTool = 'wbijajaca' THEN
	VIS.bGripperScrewer1Option3Show := FALSE;
END_IF

(****Opcja 4*****)
//Jeżeli jest włączone szukanie gwintu to kasuje szukanie gwintu w pozycji docisku
IF VIS.bGripperScrewer1FindScrewShow THEN	
	VIS.bGripperScrewer1Option4Show	:=	FALSE;	// Szukanie gwintu w pozycji dociskania
END_IF

(****Opcja 5*****)
IF NOT VIS.bGripperScrewer1FindScrewShow AND NOT VIS.bGripperScrewer1Option4Show THEN
	VIS.bGripperScrewer1Option5Show	:=	FALSE;	// Szukanie gwintu z czujnikiem wysokości
END_IF

(****Opcja 6*****)
IF VIS.lrGripperScrewerPushingCapPositionShow	= VIS.lrGripperScrewerScrewingCapPositionShow	OR 
	lrGripperScrewerPushingCapPosition			= lrGripperScrewerScrewingCapPosition OR  
	VIS.bGripperScrewer1Option5Show	OR 
	VIS.bGripperScrewer1Option4Show  //Jak jest szukanie gwintu w pozycji dociskania to nie ma ruchu od pozycji dociskania do zakrecania bo najpierw idzie do szukania
THEN
	VIS.bGripperScrewer1Option6Show := FALSE; // Obrót podczas przejścia z pozycji docisku
END_IF
END_ACTION

ACTION aStoper:
(*
fbStoperSensorDelay.bIN := P10_GripperScrewer.fbGripperScrewersDragStation.eRunningState = E_DragStationState.eDraging 
						   AND ((P00_PackML.fbPMLAuto.ePMLState = E_PMLState.ePMLState_STOPPING) OR  (P00_PackML.fbPMLAuto.ePMLState = E_PMLState.ePMLState_EXECUTE));

fbStoperSensorDelay(tFilterTimeOn:=T#120MS, tFilterTimeOff:=T#20MS);

(*tpStoperTimerOn(In:=fbStoperSensorDelay.bOUT , PT:=T#125MS);
tpStoperTimerOn.ET;

Przypisanie wyjścia z timera do wejścia na wyspę 
QbStoperActuatorOn:=tpStoperTimerOn.Q;*)
(*QbStoperActuatorOn		:= fbStoperSensorDelay.bOUT   
					  	   AND P10_GripperScrewer.fbGripperScrewersDragStation.lrActualDragPosition > P10_GripperScrewer.fbGripperScrewersDragStation.lrLeadActuatorMoveUpPosition
						   AND P10_GripperScrewer.fbGripperScrewersDragStation.lrActualDragPosition < 100;
						   
					   *)
					   
lrStoperPosition :=	(188.25 * EXPT(lrBottleDragingStationVelocity,-0.404));


tofQbGripperScrewerStoperActuator	(IN:=fbStoperSensorDelay.bOUT   AND
									P10_GripperScrewer.fbGripperScrewersDragStation.lrActualDragPosition > (lrStoperPosition+10) AND 
									P10_GripperScrewer.fbGripperScrewersDragStation.lrActualDragPosition < 100, PT:=T#500MS);
										
QbGripperScrewerStoperActuator		:= tofQbGripperScrewerStoperActuator.Q ;

(*QbGripperScrewerStoperActuator	:=	fbStoperSensorDelay.bOUT   AND
									P10_GripperScrewer.fbGripperScrewersDragStation.lrActualDragPosition > (lrStoperPosition+10) AND 
									P10_GripperScrewer.fbGripperScrewersDragStation.lrActualDragPosition < 100;*)

*)
//Manual
rtManualMode	(CLK:=bManualMode,	Q=>);
ftManualMode	(CLK:=bManualMode,	Q=>);
IF rtManualMode.Q THEN
	bGripperScrewerStoperActuatorLastState	:=	QbGripperScrewerStoperActuator;
	VIS.bGripperScrewerStoperManualActuator	:=	QbGripperScrewerStoperActuator;
END_IF
IF bManualMode THEN
	QbGripperScrewerStoperActuator		:=	VIS.bGripperScrewerStoperManualActuator;
END_IF
IF ftManualMode.Q THEN
	QbGripperScrewerStoperActuator		:= bGripperScrewerStoperActuatorLastState;
END_IF
// Koniec Manual
END_ACTION

END_PROGRAM

// ---- POUs/FB/FB_2GripperScrewers.TcPOU
(*
Nazwa:			FB_2GripperScrewers
Opis:			Zakręcarki szczekowe
Wersja:			v2.91
Data:			2026-01-12
Autor:			DP
Urzadzenia:		Serwo podnośnika, Serwo zakręcania
Ostatnie zmiany:
	- 2026-01-12 [DP] Wejście pod pozycje szukania gwintu
	- 2025-09-04 [DP] EventLog-do sprawdzenia->wywołać błędy , Estop ErrHan
	- 2025-07-09 [DP] wysokosc narzedi
	- 2025-07-08 [DP] tonError bo kasuje mcStop, tool height do błędu, opis, Resseting, Homing false w Manual
	- 2025-05-15 [DP] Zmiana errlowscrewing na -25
	- 2025-04-18 [DP] Zmiana limitu na 0.1 fullscr
	- 2025-03-31 [DP] Case 10 cofanie
	- 2025-03-31 [DP] Zmiana limitu lrPackageTurnoversToFullScrewed 0.3
	- 2025-01-17 [DP] TorqueCV 
	- 2024-12-13 [DP] Zmiany dla glowicy zasysajcej na sloiki, przejcie do pushing itd
	- 2024-12-12 [DP] Zmiana szukania gwintu
	- 2024-12-11 [DP] Skaling czuj. wysokości
	- 2024-11-26 [DP] Gear Vel sloiki
	- 2024-10-25 [DP] Zmiany torque
	- 2024-08-29 [DP] Wbijak
	- 2024-03-18 [DP] Zmiana symulacji
	- 2024-03-06 [DP] Aktualizacja instrukcji
	- 2024-02-27 [DP] Height Vel z 0 na zadaną w ressetingu, opis problemów
	- 2023-11-24 [DP] Pop. uwag dodatkowych opcji, tryb momentowy - opis
	- 2023-11-10 [DP] Akt. instrukcji, szukanie z UJL
	- 2023-03-25 [DP] przyśpieszenie screwera na stałe, zmiana instrukcji konfiguracji, skrocona czasowka griper
	- 2023-03-21 [DP] dodana ScrewerSet2
	- 2023-02-22 [DP] poprawa w GearRatio
	- 2023-02-21 [DP] Acc, Dec, Jerk i Prędkości Liftera zmniejszone 2x przez inny montaż,
				EStop w StateError, zmiana przekadni obrotu, CycleDone jak SetTorque=0,
	- 2023-02-14 [DP] Zmiana instrukcji konfiguracji
	- 2023-02-14 [DP] Wersja z LU208 z aktualizacjami z XTSa (gearing przy zakręcaniu i szukanie gwintu)
	
Konfiguracja:

Parametryzacja bloczka:
	- ustawić wysokości narzędzi, potrzebne do kolizji
	- ustawić wartość minimalną, od aktualnej wysokości zakręcarki
	

Czujnik wysokości:
	- Najlepiej przeskalować do na wejście tak, żeby pokazywał ugięcie sprężyny od transportera czyli 0mm-nieugięta
	14mm - ugięta maksymalnie (P10_GripperScrewer.IlrGripperScrewer1HeightCV:=-0.0023*(iIABPneumaticEB5AnalogueInput1)+52.006 + 1.83);

Szukanie gwintu z czujnikiem wysokości:
Włączone szukanie gwintu w pozycji dociskania i z czujnikiem wysokości, należy ustawić duży kąt obrotu (maxymalny dla szukania gwintu)
	1. Start obrotu z prędkością zadaną zakręcania, zapisywanie wartości max i min ugięcia sprężyny
	2. Szukanie 1 uskoku po 100st. o 0,5mm od wartości max ugięcia, jeżeli krotność gwintu 1x to przejście do punktu 4
	3. Szukanie 2 uskoku po 100st. jeżeli znaleziono pierwszy o 0,5mm od wartości max ugięcia
	4. Przejazd o 30,60,90st. dalej, zależnie od krotności
	5. Przejście do pozycji zakręcania lub dociskania zależnie od nastaw
	
	
Oś Obrótu (AM8031-0C20-0000): 

	Drive:
	- LU207,UBL50 - Nowa zębatka ma 32 na 48 zęby 240:360
	- ustawić driva na 'Rotatory' 360 st. i gear ratio 240:360, 240 st. na obr.
	- Invert Nc-Enc i Nc-Drive włączone
	- włączyć w drivie Scaling->Modulo data storage source - Feeback 1
	- ustawić drive Scaling->position offset setting 0 stopni na odpowiedniej pozycji na enkoderze
	- wgrać z drive Save NC parameters
	- w drivie jeszcze raz ustawić parametr Following error window 359?	
	- ustawic regulator Position mode na Kv na 10, Kp na 0.2, Tn na 0.002 
	- ustawić Acceleration Feed forward  K = 1 i wpisać inercje w Vel contr.->Vel. calc->0.001 kg m^2 oraz Mode->Basic_for_know_interia
	- ustawić w parametrach Configured channel peak current na 5A
	- ustawić w parametrach 0x6072 Bipolar torque/force limit value na 500%
	- ustawić w parametrach 0x60E0 Positive torque/force limit value na 500%
	- ustawić w parametrach 0x60E1 Negative torque/force limit value na 500%
	- dodać parametry Bipolar torque/Force limit w Process data/Outputs i polinkować ze zmienną
	- dodać parametr Positon control proportional gain Process data/Outputs i polinkować ze zmienną
	NC:
	- Ustawić Maximum Velocity na 13397.8, Reference Velocity na 14737.5, Max Acc i Dec na 300000.0
	- Default Acc i Dec na 20096.7, jerk na 60290.0
	- wyłączyć Limity Switche
	- wyłączyć wszystkie opcje Monitoringu

	Opcja trybu momentowego osi zakręcania (tylko od wersji driva 104)
	Drvie:
	- Na jednym drivie nie może być razem obrót 1 i obrót 2
	- W drivie (kanał) osi obrotu Advanced->Slots settings zaznaczyć 'I know what I do'
	i ustawiąc VelocityControlSlot na VelocityControl2, w tym momencie w IO powinny pojawić się 
	nowe wejścia,wyjścia VelocityControl2
	- W drivie Advanced->Process data rozwinąć 'Ch A Modes of operation' i ustawić '..mode_CST (10)'
	w Virual operation mode 0 
	- W parametr list powinien być parametr 0x60CA Ch a Torque limitation option code -> ustwić na
	TorqueMightBeReducedToZero, jeżeli nie ma to znaczy że trzeba zaktualizować driva lub dodać parametry ręcznie
	NC:
	- W NC w Drive->Zakładka Time Comensation-> Parametr Time Compensation Mode Drive -> 'ON(with velocity)'
	- W NC w Enc->Zakładka Time Comensation-> Parametr Time Compensation Mode Drive -> 'ON(with velocity)'
	
Oś podnoszenia (AM8032-0E21-0000):
	Drive:
	- ustawić driva na 'Linerary' 10mm i gear ratio 1:1, 10mm na obr.
	- Invert Nc-Enc i Nc-Drive włączone
	- ustawic regulator Position mode na Kv na 1, Kp na 0.2, Tn na 0.002 
	- ustawić Feed forward acceleration K = 1 i wpisać inercje w Vel contr.->Cel. calc->0 kg m^2
	NC:
	- Ustawić Maximum Velocity na 1094
	- Default Acc i Dec na 100000, jerk na 500000
	- ustawić Limit Swtiche
	- ustawić ManualVelocity (Slow) na 30 ze względu na Jog i bazowanie

Info: 
	- możliwość pracy 1 lub 2
	- możliwość pracy bez kręcenia jeżeli ustawi się prędkość 0
	- możliwosć dodatkowego chwytania przed zakręcaniem
	- step mode dla wizualizacji
	- rozróżnienie warningów

Tryb momementowy:
lrPackageTurnoversToFullScrewed - Ilośc obrotów do zakręcenia
iScrewer1SetTorque - Zadany moment w % (Przeliczany z Nm z wizualizacji)
lrScrewerSpeed - Prędkość zakręcania w st/s (Przeliczany z rpm z wizualziacji)
1. Start											Rozpędzanie,	Torque 5000 (Max) [%], 				TorqueRamp 4000 [%/s], VelocityLimitLow -5000 (Max) [st./s]
2. ActPos>lrPackageTurnoversToFullScrewed*360.0/7	Hamowanie,		Torque -9 [%],						TorqueRamp 1500 [%/s], VelocityLimitLow -4000 (Max) [st./s]
3. ActPos>lrPackageTurnoversToFullScrewed*360.0/6	Dokręcanie,		Torque iScrewer1SetTorque [%],		TorqueRamp 4000 [%/s], VelocityLimitLow lrScrewerSpeed (Max) [st./s]



Jak naprawić:
A. Zakręcarka nie wykonuje ruchu w trybie momentowym, jedna działa , druga nie - sprawdzić czy bloczek MC_Torque wykonuje ruchu,
jeżeli nie to wyłączyć VelocityControl2, włączyć bez '2' i ponownie włączyć '2', potem aktywacja
B. 
*)

FUNCTION_BLOCK FB_2GripperScrewers
VAR_INPUT
	bEnable1							:BOOL;		//Zezwolenie na pracę 1
	bEnable2							:BOOL;		//Zezwolenie na pracę 2
	bEstop								:BOOL;		//Stop awaryjny nieaktywny
	bRun1								:BOOL;		//Rozkaz zakręcania zakręcarki 1
	bRun2								:BOOL;		//Rozkaz zakręcania zakręcarki 2
	bSimulation							:BOOL;		//Włączona symulacja, skracanie czasu przerywania jak nie ma butelki
	bHoming								:BOOL;		//Zezwolenie na wykonanie bazowania i pozycjonowania zakręcarki
	bHeightSet							:BOOL;		//Ustaw wysokość
	bIgnoreError						:BOOL;		//Ignorowania błędów cyklu pracy
	bScrewer1SetPositionOffset			:BOOL;		//Ustaw offset obrotu zakręcarki 1
	bScrewer2SetPositionOffset			:BOOL;		//Ustaw offset obrotu zakręcarki 2
	iScrewer1AddTorque					:UINT;
	iScrewer2AddTorque					:UINT;
	bReset								:BOOL;		//Reset błędu, jeśli w stanie "eError
	iTool								:INT;		// Wybór narzędzia (1-5), opisy w tablicy AsGripperScrewerTool	
	bOptionOpenedGripperWhenFindingScrew:BOOL;		//OPCJA. Otwarty chwytak przy szukaniu gwintu
	bOptionScrewingBackwardsInPushingPosition:BOOL;	//OPCJA. Obrót do tyłu w pozycji dociskania
	bOptionCapPushingWithoutScrewing	:BOOL;		//OPCJA. Tylko wbijanie bez zakręcania
	bOptionCapPositioning				:BOOL;		//OPCJA. Dodatkowe zamknięcie chwytakiem przed zakręceniem (do testów)
	bOptionFindScrewInScrewingPosition	:BOOL;		//OPCJA. Szukaj początku gwintu nakrętki i opakowania. Zakręcarka napjpierw obraca się w lewo, a po znalezienu gwintu przystepuje do zakręcania w pozycji zakręcania
	bOptionFindScrewInPushingPosition	:BOOL;		//OPCJA. Szukaj początku gwintu nakrętki i opakowania. Zakręcarka napjpierw obraca się w lewo, a po znalezienu gwintu przystepuje do zakręcania w pozycsji docisku
	bOptionFindScrewWithHeightSensor	:BOOL;		//OPCJA. Szukanie gwintu z czujnikiem wysokości
	bOptionFindScrewRotateFromPushingToScrewingSensor	:BOOL;		//OPCJA. Obrót od pozycji docisku do zakręcania
	bOptionMomentaryMode				:BOOL;		//OPCJA. Tryb momentowy zakręcania
	lrPackageTurnoversToFullScrewed		:LREAL;		//Obroty do pełnego zakręcenia
	lrPackageThreadPitch				:LREAL;		//Skok gwintu
	lrPackageThreadTimes				:LREAL;		//Krotność gwintu
	lrHeightReadyPosition				:LREAL;		//Wysokość zadana w stanie gotowości od płyty[mm]
	lrHeightPushingPosition				:LREAL;		//Wysokość zadana przy wciskaniu nakrętki od płyty[mm]
	lrHeightEndScrewingPosition			:LREAL;		//Wysokość zadana przy zakręcaniu nakrętki od płyty [mm]
	lrHeightFindScrewPosition			:LREAL;		//Pozycja szukania gwintu [mm]
	lrHeightScrewingDistanceSpeed		:REAL;		//Prędkość obniżania podczas zakręcania
	lrHeightActualPosition				:LREAL;		//Aktualna pozycja podnośnika
	lrSpringHeightCV					:LREAL;		//Czujnik ugięcia sprężyny (przeskalować na 0-14mm (14mm-maksymalnie ugięta)
	lrHeightActualTorque				:LREAL;		//Aktualny moment [%]
	rActualMotor1Temperature			:REAL;		//Aktualna temperatura silnika 1
	rActualMotor2Temperature			:REAL;		//Aktualna temperatura silnika 2
	iHeightSetTorque					:INT;		//Zadany moment dociskania [%]
	iScrewer1SetTorque					:INT;		//Zadany moment dokręcania [%]
	iScrewer2SetTorque					:INT;		//Zadany moment dokręcania [%]
	iScrewTightTime						:INT;		//Czas przytrzymania po uzyskaniu momentu [ms] 
	lrScrewer1ActualTorque				:LREAL;		//Aktualny moment [%]
	lrScrewer2ActualTorque				:LREAL;		//Aktualny moment [%]
	lrHeightAcceleration				:LREAL;		//Przyspieszenie podnosnika zakręcarki
	lrHeightDeceleration				:LREAL;		//Opóźnienie podnośnika zakręcarki
	lrHeightSpeed						:LREAL;		//Prędkość podnośnika zakręcarki
	lrScrewer1ActualPosition			:LREAL;	
	lrScrewer2ActualPosition			:LREAL;	
	lrScrewerAcceleration				:LREAL;		//Przyspieszenie zakręcania
	lrScrewerDeceleration				:LREAL;		//Opóźnienie zakręcania
	lrScrewerSpeed						:LREAL;		//Prędkość zakręcania
	lrScrewer1PosDiff					:LREAL;		//ScrewingAxisRef.NcToPlc.PosDiff
	lrScrewer2PosDiff					:LREAL;		//ScrewingAxisRef.NcToPlc.PosDiff
	lrFindigScrewDegree					:LREAL;		//Kąt wycofania zakręcarki przy szukaniu gwintu
	bManualMovement						:BOOL;		//Zezwolenie na ruchy ręcznę
	lrManualOverride					:LREAL;		//Procentowa redukcja prędkości wszystkich serw (Tylko w trybie manualnym)
                                	
	lrMaxHeightPosition:LREAL;				//Wysokość maksymalna zakręcarki 
	lrMinHeightPosition:LREAL;				//Wysokość minimalna zakręcarki 
	lrMaxScrewerSpeed	:LREAL;				//Maksymalna prędkość zakręcania

	//StepMode
	bStepMode				: BOOL;		//Włączony tryb skokowy sterowania podnośnikami (tylko w serwisie)
	lrSetPosStepMode		: LREAL; 	//Ruch podnośnika o zadaną wartość w trybie krokowym (tylko w serwisie)
	
	_ALARMINFO_ :BOOL;
	iStationIndex:UDINT;					//Numer stacji 
	sStationName:WSTRING;					//Nazwa stacji
END_VAR

VAR_OUTPUT
	eState							: E_Station;				//Stan ogólny bloku
	eRunningState					: E_GripperScrewer; 		//Stan zakręcarki
	bError							: BOOL;						//Błąd stacji
	udiErrorID						: UDINT;					//Nr błędu zakręcarki
	sErrorDescription				: STRING(200);				//Opis błędu
	sErrorDescription2				: STRING(200);				//Opis błędu
	sErrorStationName				: STRING;					//Nazwa stacj
	udiStationID					: UDINT;				// Nr stacji
	
	udiHeightServoErrorNr			: UDINT;					//Nr błędu serwo podnośnika
	udiScrewing1ServoErrorNr		: UDINT;					//Nr błędu serwo zakręcarki 1
	udiScrewing2ServoErrorNr		: UDINT;					//Nr błędu serwo zakręcarki 2
	bGripper1Actuator				: BOOL;						//Siłownik chwytaka
	bGripper2Actuator				: BOOL;						//Siłownik chwytaka
	uiScrewing1TorqueControl		: UINT;						//Kontola momentu zakręcania	
	uiScrewing2TorqueControl		: UINT;						//Kontola momentu zakręcania	
	rScrewing1ProportionalGain		: UINT;						//Kontola Kp
	rScrewing2ProportionalGain		: UINT;						//Kontola Kp	
	lrScrewer1TorqueCV				: LREAL;					//Wartość osiągniętego momentu dokręcenia [nM]
	lrScrewer2TorqueCV				: LREAL;					//Wartość osiągniętego momentu dokręcenia [nM]
	uiHeightTorqueControl			: UINT						:= 6000;
	sWarningDescription				: STRING;
	bWarning1						: BOOL;
	bWarning1A						: BOOL;	
	bWarning1B						: BOOL;	
	bWarning1C						: BOOL;	
	bWarning1D						: BOOL;	
	bWarning1E						: BOOL;	{warning'dorobic ostrzezenie szukania gwintu}
	bWarning2						: BOOL;
	bWarning2A						: BOOL;	
	bWarning2B						: BOOL;	
	bWarning2C						: BOOL;	
	bWarning2D						: BOOL;	
	bWarning2E						: BOOL;	
	udiWarningID					: UDINT;
	tCycleTime						: TIME;	
	bHomingDone						: BOOL;						//Wymagane ponowne bazowanie (blad podczas bazowania lub stop awaryjny)
	bCycleDone1						: BOOL;
	bCycleNotDone1					: BOOL;		
	bCycleDone2						: BOOL;
	bCycleNotDone2					: BOOL;		
	bAdjustingTorqueDone			: BOOL;
	iAdjustingTorque				: INT;
	lrAdjustingMaxTorque			: LREAL;
	AsToolDescription				: ARRAY [0..10] OF STRING;	// Opis narzędzi, 1 - Opis narzędzia nr 1, 2 - Opis narzędzia nr 2
	sTool							: STRING;
	iToolHeight						: INT;	//Wysokość narzędzia od dolnej metalowej częsci dwuszczekowego
END_VAR

VAR_IN_OUT
	bManualHeightUp					:BOOL;			//Ruch ręczny podnośnikiem stacji w górę
	bManualHeightDown				:BOOL;			//Ruch ręczny podnośnikiem stacji w dół
	bManualScrew1Clockwise			:BOOL;			//Ruch ręczny zakręcarką w kierunku wskazówek zegara;
	bManualScrew1CClockwise			:BOOL;			//Ruch ręczny zakręcarką w kierunku przeciwnym do wskazówek zegara;
	bManualScrew2Clockwise			:BOOL;			//Ruch ręczny zakręcarką w kierunku wskazówek zegara;
	bManualScrew2CClockwise			:BOOL;			//Ruch ręczny zakręcarką w kierunku przeciwnym do wskazówek zegara;
	bManualGripper1					:BOOL;			//Ruch zamknięcie chwytaka nakrętek
	bManualGripper2					:BOOL;			//Ruch zamknięcie chwytaka nakrętek
	HeightAxisRef					:AXIS_REF;		//Struktura sterowania NC dla serwa podnoszenia zakręcarki
	Screwing1AxisRef				:AXIS_REF;		//Struktura sterowania NC dla serwa zakręcania
	Screwing2AxisRef				:AXIS_REF;		//Struktura sterowania NC dla serwa zakręcania	
	bFindScrewAdjustSensorHeight	:BOOL;			//Włacz szukanie MIN i MAX jeżeli jest opcja z czujnikie wysokości
	bAdjustingTorque				:BOOL;			//Dobieranie momentu
	lrAdjustingSetTorque			:LREAL;	
END_VAR

VAR
	bScrew1Found					: BOOL; 						// Zakręcarka znalazła początek gwintu
	bScrew2Found					: BOOL; 						// Zakręcarka znalazła początek gwintu	
	tonTightScrewing1Timer			: TON; 							// Timer potwierdzenia dokręcenia nakrętki
	tonTightScrewing2Timer			: TON; 							// Timer potwierdzenia dokręcenia nakrętki
	tonTightScrewing1TimerAndOpenedGripper	: TON; 					// Timer potwierdzenia dokręcenia nakrętki
	tonTightScrewing2TimerAndOpenedGripper	: TON; 					// Timer potwierdzenia dokręcenia nakrętki	
	tonMomentaryScrewing1Timer		: TON; 							// Timer potwierdzenia dokręcenia nakrętki
	tonMomentaryScrewing2Timer		: TON; 							// Timer potwierdzenia dokręcenia nakrętki

	bScrewed1					: BOOL; 						// Nakrętka zakręcona
	bScrewed2					: BOOL; 						// Nakrętka zakręcona
	tonTooLongScrewing1			: TON;							// Błąd zbyt długiego zakręcania
	tonTooLongScrewing2			: TON; 							// Błąd zbyt długiego zakręcania	
	tTooLongScrewing1			: TIME;							// Czas  zbyt długiego zakręcania
	tTooLongScrewing2			: TIME; 						// Czas  zbyt długiego zakręcania		
	tonGripper1ReliseDelay		: TON;							// Time Opóźniajacy ruch w górę po zakręceniu, pozwalajac na otwarcie chwytaka
	tonGripper2ReliseDelay		: TON;							// Time Opóźniajacy ruch w górę po zakręceniu, pozwalajac na otwarcie chwytaka
	tonGripper1ReliseDelay2		: TON;							// Time Opóźniajacy ruch w górę po zakręceniu, pozwalajac na otwarcie chwytaka
	tonGripper2ReliseDelay2		: TON;							// Time Opóźniajacy ruch w górę po zakręceniu, pozwalajac na otwarcie chwytaka

	mcScrewer1ManualMove		: MC_JOG; 						// Blok obrotu ręcznego zakręcarką
	mcScrewer2ManualMove		: MC_JOG; 						// Blok obrotu ręcznego zakręcarką
	mcScrewer1Stop				: MC_Stop;						// Trwałe zatrzymywanie Serwo
	mcScrewer2Stop				: MC_Stop;						// Trwałe zatrzymywanie Serwo
	mcScrewer1MoveVelocity		: MC_MoveVelocity;				// Ruch prędkościowy
	mcScrewer2MoveVelocity		: MC_MoveVelocity;				// Ruch prędkościowy
	mcScrewer1MoveVelocity2		: MC_MoveVelocity;				// Ruch prędkościowy
	mcScrewer2MoveVelocity2		: MC_MoveVelocity;				// Ruch prędkościowy
	mcScrewer1MoveVelocity3		: MC_MoveVelocity;				// Ruch prędkościowy
	mcScrewer2MoveVelocity3		: MC_MoveVelocity;				// Ruch prędkościowy	
	mcScrewer1MoveRelative		: MC_MoveRelative; 				// Ruch relatywny zakręcarki
	mcScrewer2MoveRelative		: MC_MoveRelative; 				// Ruch relatywny zakręcarki
	mcScrewer1MoveAbsolute		: MC_MoveAbsolute; 				// Ruch absolutny zakręcarki
	mcScrewer2MoveAbsolute		: MC_MoveAbsolute; 				// Ruch absolutny zakręcarki
	fbScrewer1SetPositionOffset	: FB_CoEAX8000SetPositionOffset;// Ustawianie pozycji obrotu 
	fbScrewer2SetPositionOffset	: FB_CoEAX8000SetPositionOffset;// Ustawianie pozycji obrotu 
	mcScrewer1TorqueControl		: MC_TorqueControl;
	mcScrewer2TorqueControl		: MC_TorqueControl;
	
	mcScrewing1Power			: MC_Power;			 			// Zasilanie napędu zakręcarki
	mcScrewing2Power			: MC_Power;			 			// Zasilanie napędu zakręcarki
	bScrewer1ServoPower			: BOOL; 						// Zmienna sterujaca zasilaniem serwo Zakręcarki
	bScrewer2ServoPower			: BOOL; 						// Zmienna sterujaca zasilaniem serwo Zakręcarki
	fbScrewer1HardReset			: FB_SoEReset; 					// Blok twardego resetu serwa zakręcania
	fbScrewer2HardReset			: FB_SoEReset; 					// Blok twardego resetu serwa zakręcania
	mcScrewer1SoftReset			: MC_Reset; 					// blok łagodnego resetu serwa zakręcarki
	mcScrewer2SoftReset			: MC_Reset; 					// blok łagodnego resetu serwa zakręcarki
	
	mcHeightManualMove			: MC_JOG; 						// Blok sterowania ręcznego wysokością
	mcHeightStop				: MC_STOP; 						// Trwałe Zatrzymywanie ruchu podnośnika zakręcarki
	mcHeightMoveAbsolute		: MC_MoveAbsolute;				// Blok sterowania wysokością	
	mcHeightPower				: MC_POWER; 					// Uruchomienie zasilania serwa podnosnika zakręcarki
	bHeightServoPower			: BOOL; 						// Zmienna sterowania zasilaniem serwo
	fbHeightHardReset			: FB_SoEReset; 					// Blok Twardego resetu serwa podnośnika zakręcarki
	mcHeightSoftReset			: MC_Reset; 					// Blok łagonego resetu podnośnika zakręcarki
	mcHeightGearInMultiMaster	: MC_GearInMultiMaster; 		// Blok sprzęgania podnoszenia z zakręcaniem
	mcHeightGearOut				: Mc_GearOut;					// Blok wysprzeglania podnoszenia z zakręcaniem

	(*Axis online*)
	fbHeight					: FB_McAxisOnlineAX8000;
	stHeight					: ST_McAxisOnline;
	fbScrewing1					: FB_McAxisOnlineAX8000;
	stScrewing1					: ST_McAxisOnline;
	fbScrewing2					: FB_McAxisOnlineAX8000;
	stScrewing2					: ST_McAxisOnline;
	
	(*Ostrzezenia,przerywanie*)
	tonTooLongFinding1			: TON; 							// Za długie szukanie gwintu
	tonTooLongFinding2			: TON; 							// Za długie szukanie gwintu
	tonPosDiff1Error			: TON;
	tonPosDiff2Error			: TON;
	tonPosTooLowWhenScrewing1	: TON;
	tonPosTooLowWhenScrewing2	: TON;
	
	(*Statistics*)
	tonCycleTimer				: TON;
	rtrigCycleTimerRead			: R_TRIG;

	lrStartPosition1			: LREAL;
	lrStartPosition2			: LREAL;
	tonMaxHeight				: TON;

	tonGripper1Delay			: TON;
	tonGripper2Delay			: TON;
	
	eLastState					: E_Station;			// Stan ogólny bloku
	eLastRunningState			: E_GripperScrewer;		// Stan podbloku
	eLastStateTemp				: E_Station;			// Stan ogólny bloku
	eLastRunningStateTemp		: E_GripperScrewer;		// Stan podbloku

	bStateError: BOOL;
	bHeighSetNotDone: BOOL;
	
	(*Szukanie momentu*)
	nCaseAdjustingTorque					: INT;
	tonAdjustingTightScrewingTimer			: TON;
	tonAdjustingGripperClose				: TON;
	uiAdjustingScrewerTorqueControl			: UINT;
	bAdjustingScrewed						: BOOL;
	tonAdjustingCase40						: TON;
	bAdjustingSetTorqueAchieved				: BOOL;
	bAdjustingTorqueTooHigh					: BOOL;
	bAdjustingTorqueTooLow					: BOOL;
	lrMotorNominalTorque					: LREAL;
	lrScrewerActualTorqueNm					: LREAL;
	
	tonFindingScrew						: TON;
	tonScrew1Found						: TON;
	tonScrew2Found						: TON;
	tonDelayServoOn						: TON;

	bPreparingToDisable					: BOOL;
	bHeightGearingWithScrewer			: BOOL;
	iStoppingCase						: INT;
	iScrewingCase						: INT;
	iScrewing2Case						: INT;
	
	(*Bledy, Resetowanie*)
	tonResetting						: TON;
	tonEstop							: TON;
	tonError							: TON;	
	rtResetCommands						: R_TRIG;
	tonActualMotor1TemperatureTooHigh	: TON;
	tonActualMotor2TemperatureTooHigh	: TON;
	iErrorResseting3					: INT;
	iTestError3							: INT;
	iTestError4							: INT;
	
	(*Metoda*)
	mcMoveAbsolute						: MC_MoveAbsolute; 				// Ruch absolutny
	iMStep								: INT;							// Do testów
	bPrepareToReadyTest					: BOOL;							// Do testów	

	(*Bazowanie*)
	iHomingCase							: INT;
	iPreparingToReadyCase				: INT;
	
	(*Czytanie momentu*)
	rtRun1								: R_TRIG;
	rtRun2								: R_TRIG;

	(*Step Mode*)
	rtStepModeUp						: R_TRIG;
	rtStepModeDown						: R_TRIG;
	lrStepModeHeightMotorSV				: LREAL;
	bStepModeMoving						: BOOL;
	tofStepModeMoving					: TOF;	
	
	(*Running*)
	iGoingUpCase						: INT;
	iToPushingPositionCase				: INT;
	tonDelayBeforeResetLag				: TON;
	lrGearRatio1						: LREAL;
	lrGearRatio2						: LREAL;
	lrSf1								: LREAL;	
	lrSf2								: LREAL;
	lrDivider							: LREAL;	
	
	(*Dodatkowe chwytanie przed zakreceniem*)
	iCloseGripperBeforeScrewingCASE		: INT;
	
	(*Bez zakręcania*)
	tonHoldingTimer						: TON;
	
	(*Aborting*)
	iAbortingCASE						: INT;
	
	(*Szukanie gwintu*)
	iFindingScrewCASE							: INT;
	lrScrewer1MaxTorqueWhenFindingScrew			: LREAL; //OPCJA 1
	lrScrewer2MaxTorqueWhenFindingScrew			: LREAL; //OPCJA 1	
	lrScrewerMinTorqueWhenFindingScrew			: LREAL; //OPCJA 1
	lrScrewerMaxSensorHeightWhenFindingScrew	: LREAL:= -100000; //OPCJA 2
	lrScrewerMinSensorHeightWhenFindingScrew	: LREAL:= 0; //OPCJA 2
	bScrew1MinFound								: BOOL;
	bScrew2MinFound								: BOOL;
	lrStartPosition1FindingScrew				: LREAL;
	lrStartPosition2FindingScrew				: LREAL;
	lrFindingScrewPositionDelay					: LREAL;	
	tonFindingScrewDelay						: TON;
	iFindScrewAdjustSensorHeight				: INT;
	
	(*Symulacja*)
	tonSimulationScrewing1						: TON;
	tonSimulationScrewing2						: TON;	
	
	(*inne*)
	iTestResetting: INT;
	iCountAborting: INT;
	bTest2:BOOL;
	lrScrewerOffsetSensorHeightWhenFindingScrew: LREAL;
	bTest: BOOL;
	iTesty: INT;
	tonTesty1: TON;
	tonTesty2: TON;	
	
	//Zmienne od EVENTLOGGER
	bAlarmInit 						: BOOL := TRUE; 
	nAlarmNumerator					: INT;
	arfbAlarm						: ARRAY[0..19] OF  FB_TcAlarm;		//Tablica bloczków błędów
	fbSourceInfo 					: FB_TcSourceInfo;
	iSourceInfo						: I_TcSourceInfo;
	sAlarmTest						: STRING;
	//Koniec zmiennych od EVENTLOGGER
	
END_VAR

IF bPrepareToReadyTest THEN
	IF	M_PrepareToReady(	AxisRef			:=  Screwing1AxisRef,			
                   			iGripperArms	:=	2
						)	
	THEN
		bPrepareToReadyTest := FALSE;
	END_IF			
				   
END_IF  

//Wywołanie AXIS Online
(*fbHeight	(stMcAxisOnline:= stHeight,		Axis:= HeightAxisRef);
fbHeight	(stMcAxisOnline:= stHeight,		Axis:= HeightAxisRef);
fbScrewing1	(stMcAxisOnline:= stScrewing1,	Axis:= Screwing1AxisRef);
fbScrewing1	(stMcAxisOnline:= stScrewing1,	Axis:= Screwing1AxisRef);
fbScrewing2	(stMcAxisOnline:= stScrewing2,	Axis:= Screwing2AxisRef);
fbScrewing2	(stMcAxisOnline:= stScrewing2,	Axis:= Screwing2AxisRef);
*)
//Parametryzacja
bHeightGearingWithScrewer := TRUE;

Tools();
ErrorHandling();
Control();
Limits();
AdjustingTorque();
HeightControlBlocks();
TorqueControl();
Screwer1ControlBlocks();
Screwer2ControlBlocks();
Simulation();
ReadScrewingTorque();
Statistics();
Warnings();
aStationID();
aTesty();
(*Zapisywanie ostatniego stanu*)
IF eLastStateTemp<>eState THEN
	eLastState := eLastStateTemp;
END_IF
eLastStateTemp := eState;
IF eLastRunningStateTemp<>eRunningState THEN
	eLastRunningState := eLastRunningStateTemp;
END_IF
eLastRunningStateTemp := eRunningState;
(*Koniec Zapisywanie ostatniego stanu*)


(*Dodatkowe zabezpieczenie przed uderzeniem w chwytak*)
IF mcHeightMoveAbsolute.Execute AND (mcHeightMoveAbsolute.Position-iToolHeight)<=lrMinHeightPosition THEN
	mcHeightMoveAbsolute.Execute:=FALSE;
END_IF
	
IF mcHeightMoveAbsolute.Error THEN
	mcHeightMoveAbsolute.Execute:=FALSE;
END_IF

IF mcScrewer1MoveVelocity.Error THEN
	mcScrewer1MoveVelocity.Execute:=FALSE;
END_IF	
(*Koniec dodatkowe zabezpieczenie przed uderzeniem w chwytak*)


(*Zabezpieczenie przed kolizją stacji poprzez ruch podnośnika*)	
IF bManualHeightDown AND (HeightAxisRef.NcToPlc.ActPos-iToolHeight)<=lrMinHeightPosition AND NOT bHoming AND NOT bHeightSet THEN
	bManualHeightDown:=FALSE;
END_IF	

IF bManualHeightUp AND (HeightAxisRef.NcToPlc.ActPos)>=lrMaxHeightPosition AND NOT bHoming AND NOT bHeightSet THEN
	bManualHeightUp:=FALSE;
END_IF	
(*Koniec zabezpieczenia przed kolizją stacji poprzez ruch podnośnika*)

ACTION AdjustingTorque:
(*

bAdjustingTorque;								// Wlączenie szukania 
lrAdjustingSetTorque;							// Szukany moment [Nm]
uiAdjustingScrewerTorqueControl; 				// Badanie tym momentem, zwiekszanie o ileś
lrMotorNominalTorque					:=	3.192; 		

tonAdjustingGripperClose		(IN:=	bGripper1Actuator, 																		PT:=T#200MS);
tonAdjustingTightScrewingTimer	(IN:=	nCaseAdjustingTorque = 30 AND (lrScrewer1ActualTorque>=uiAdjustingScrewerTorqueControl),	PT:=T#1000MS);
tonAdjustingCase40				(IN:=	nCaseAdjustingTorque=40,																PT:=T#200MS);

CASE nCaseAdjustingTorque OF
	
	0: //Włączanie
		IF bAdjustingTorque AND NOT bAdjustingTorqueDone THEN
			//Kasowanie zmiennych
			lrStartPosition1				:=	0;
			uiAdjustingScrewerTorqueControl	:=	0;
			iAdjustingTorque				:=  0;
			lrAdjustingMaxTorque			:= 	0;
			bAdjustingTorqueTooHigh			:=	FALSE;
			bAdjustingTorqueTooLow			:=	FALSE;
			nCaseAdjustingTorque			:=	10;
			mcScrewer1MoveVelocity.Execute	:=	FALSE;
		END_IF
		
	10: //Zamykanie chwytaka
		bGripper1Actuator					:=	TRUE;
		IF tonAdjustingGripperClose.Q THEN
			nCaseAdjustingTorque			:=	20;
		END_IF
		
	20:	//Ustawienie dużego momentu na początek ruchu
		uiScrewing1TorqueControl				:=  6000;
		lrStartPosition1						:=	Screwing1AxisRef.NcToPlc.ActPos;		

		IF  bAdjustingTorqueTooLow	THEN
			bAdjustingTorqueTooLow				:= FALSE;
			uiAdjustingScrewerTorqueControl		:=  uiAdjustingScrewerTorqueControl + 1;
		ELSIF bAdjustingTorqueTooHigh	THEN
			bAdjustingTorqueTooHigh				:= FALSE;
			IF uiAdjustingScrewerTorqueControl	>	0 THEN
			uiAdjustingScrewerTorqueControl		:=  uiAdjustingScrewerTorqueControl - 1;
			END_IF
		END_IF
		nCaseAdjustingTorque				:=	30;
		
	30:	 //Zakręcanie

		//Zacznij zakręcać
		lrScrewerAcceleration				:=	26000;
		lrScrewerDeceleration				:=	26000;
		mcScrewer1MoveVelocity.Direction		:=	MC_Positive_Direction;
		mcScrewer1MoveVelocity.Velocity		:=	5000;
		mcScrewer1MoveVelocity.Execute		:=	TRUE;
		
		//Zwiększanie momentu na początek ruchu
		IF ABS(ABS(lrStartPosition1)-ABS(Screwing1AxisRef.NcToPlc.ActPos))>15 OR ABS(Screwing1AxisRef.NcToPlc.PosDiff)>15  THEN 
			uiScrewing1TorqueControl			:=	(uiAdjustingScrewerTorqueControl+3)*10;
		ELSE
			uiScrewing1TorqueControl			:=	(uiAdjustingScrewerTorqueControl+3)*10+500;	
		END_IF
		
		IF tonAdjustingTightScrewingTimer.Q THEN //Jeżeli osiągnięty moment przez 200MS
			mcScrewer1MoveVelocity.Execute	:=	FALSE;
			mcScrewer1SoftReset				(Axis:=Screwing1AxisRef, Execute:= TRUE);
			iAdjustingTorque				:= UINT_TO_INT(uiScrewing1TorqueControl/10);
			uiScrewing1TorqueControl			:=	0;
			bAdjustingScrewed				:=	TRUE;		
		END_IF
			   
		IF mcScrewer1MoveVelocity.Execute = FALSE AND bAdjustingScrewed THEN
			nCaseAdjustingTorque			:=	40;
		
		END_IF	
		
	40:	//Czekanie po zakręceniu
		mcScrewer1SoftReset					(Axis:=Screwing1AxisRef, Execute:= FALSE);
		uiScrewing1TorqueControl				:=	0;
		lrStartPosition1						:=	0;
		lrAdjustingMaxTorque				:= 	0;
		bAdjustingScrewed					:=	FALSE;
		IF tonAdjustingCase40.Q THEN
			lrStartPosition1					:=	Screwing1AxisRef.NcToPlc.ActPos;	
			uiScrewing1TorqueControl			:=	1;
			nCaseAdjustingTorque			:=	50;
		END_IF
		
	50: //Odkręcanie

		lrScrewerAcceleration				:=	20;
		lrScrewerDeceleration				:=	20;
		mcScrewer1MoveVelocity.Direction		:=	MC_Negative_Direction;
		mcScrewer1MoveVelocity.Velocity		:=	10;
		mcScrewer1MoveVelocity.Execute		:=	TRUE;
		uiScrewing1TorqueControl				:=	6000;
		
		//Szukanie największego momentu w Nm
		lrScrewerActualTorqueNm:=(ABS(lrScrewer1ActualTorque)/100.0)*lrMotorNominalTorque;
		IF lrScrewerActualTorqueNm	>=	lrAdjustingMaxTorque THEN
			lrAdjustingMaxTorque			:=	lrScrewerActualTorqueNm;
		END_IF
		
		//Jeżeli osiągnięty moment
		IF lrAdjustingMaxTorque>=lrAdjustingSetTorque - 0.1 AND lrAdjustingMaxTorque<=lrAdjustingSetTorque + 0.1 THEN
			bAdjustingSetTorqueAchieved 	:= TRUE;
		ELSE
			bAdjustingSetTorqueAchieved 	:= FALSE;
		END_IF
		
		
